(* CODESYS project std12k5_8.project

Project tree, tasks and I/O mapping:
  K1 : ELNA PLC-03-02R, OOO ELNA, version 3.5.0.31
    application std12k5
      libraries: Standard, * (System); Util, * (System); CmpSchedule, 3.5.2.0 (System); CmpLog, 3.5.2.0 (System); SysCom, 3.3.2.50 (System); SysFile, 3.3.2.50 (System); SysFileAsync, 3.3.2.50 (System); SysDir, 3.3.2.50 (System); SysTimeRtc, 3.5.0.0 (System); SysTime, 3.4.1.20 (System); CAA Storage, 3.4.4.0 (CAA Technical Workgroup); SysTypes, 3.1.2.0 (System); CmpErrors Interfaces, * (System); CmpDynamicText, 3.4.1.0 (System); SysShm, 3.3.2.50 (System); SysProcess, 3.3.2.50 (System); CmpTraceMgr, 3.5.0.0 (System); 3S Storage, 3.4.4.0 (3S - Smart Software Solutions GmbH)
      task Task (cyclic, interval t#200ms, priority 1) calls MAIN
      task TaskREZ (cyclic, interval t#110ms, priority 10) calls REZERV1
      hardwareConfig/
        data type AOConfig
        defines/
          global variables hwC
        data type DOConfig
        data type AiConfig
        data type DiConfig
      logicConfig/
        defines/
          global variables logicConfig
      program MAIN [ST]
      algoritms/
        defines/
          global variables algoritmsConf
        data type AlgoritmsConfig
        data type ImConfig
        data type ModeGpa
        data type ProtectionsConfig
        data type YstavkiConfig
      modbus/
        data type MbsConfig
        function block tstModbus [ST]: ProcessInputs, ProcessOutputs
      function block AlgoritmsManager [ST]: onStart, onInit, setMode, resetAndDisable
      function block ProtectionManager [ST]: anyProtectionSignaling
      Elpk_03_02/
        program MainUP_PRG [ST]
        global variables GVL_COMMON
        global variables GVL1N_REZ
        global variables GVLOPC
        declarations NVL1_REZ
      Symbols
      Logic/
        function block PPU_Init [ST]
        function block Synch_Rejims [ST]
        function block SIP_PS [ST]
        function block All_Quation_Off [ST]
        function block AI_Final [ST]: setNewSIP
        function block AI_Final_SIP [ST]: setNewSIP
      nasos/
        function block AutoAVOM [ST]: AVOMs_Vkl, reset, AVOMs_Vykl, run
        function block AutoNuAlg_2 [ST]: reset
        function block AutoNuAlg_1 [ST]: reset
        function block AutoPnsALg [ST]: reset
        function block AutoTEN [ST]: run, reset
        function block PNS_ON_MV_ON [ST]: reset
      function block OpcCommands [ST]
      ostanov/
        function block aoAlg [ST]: reset, run
        function block noAlg [ST]: reset, run
      Prov/
        function block Opressovka [ST]: reset
        function block Prov_dPmg [ST]: reset, run
        function block Prov_Pms [ST]: reset, run
        function block Test_Protections [ST]: reset, run, Run_Protection
        function Reset_ALL_P [ST]
      Pusk/
        function block puskSecond_faza_Chastotny [ST]: run, reset
        function block ppuAlg [ST]: AS_PS_Anologs, haveAlarms, reset, writeImStatus, remont, analogsNS, CK_Di, Neisp_DI
        function block puskFirst_faza1 [ST]: reset, run
        function block puskFirst_faza2 [ST]
        function block puskSecond_faza_Reactor [ST]: reset, run
        function block puskThird_faza [ST]: reset, run
      Start_ALG/
        function block Kran_6_Close [ST]: reset
        function block Kran_6_MOVE [ST]: reset, run
        function block PNS_Pusk [ST]: reset
        function block Reset_AutoAVOM [ST]: reset
        function block Reset_AutoTEN [ST]: reset
        function block Reset_Test_IM [ST]: reset
        function block Start_AutoAVOM [ST]: reset
        function block Start_AutoTEN [ST]: reset
        function block Start_ProtectionsVibr [ST]: reset
        function block Start_Prov_dPmg [ST]: reset
        function block Start_Prov_I [ST]: reset
        function block Start_Prov_k [ST]: reset
        function block Start_Prov_Pms [ST]: reset
        function block Start_Prov_V [ST]: reset
        function block Start_Pusk_AP [ST]: reset
        function block Start_Pusk_PP [ST]: reset
        function block Start_Test_IM [ST]: reset
        function block Start_NO [ST]: reset
        function block Start_AO [ST]: reset
        function block Start_Test_Pr [ST]: reset
      TestIm/
        function BlockIm [ST]
        function BlockOpcControl [ST]
        function block TestImAlg [ST]: reset, run
        function block Imit_OPC [ST]
      Narabotka/
        function block AO [ST]: readPersistent, writePersistent
        function block Avom1 [ST]: readPersistent, writePersistent
        function block Avom2 [ST]: readPersistent, writePersistent
        function block Avom3 [ST]: readPersistent, writePersistent
        function block Avom4 [ST]: readPersistent, writePersistent
        function block EO [ST]: readPersistent, writePersistent
        function block NO [ST]: readPersistent, writePersistent
        function block nu1 [ST]: readPersistent, writePersistent
        function block nu2 [ST]: readPersistent, writePersistent
        function block pns_ [ST]: readPersistent, writePersistent
        function block Pusk [ST]: readPersistent, writePersistent
        function block Work [ST]: readPersistent, writePersistent
        function block CMN_ [ST]: readPersistent, writePersistent
        function block Kalorifer_AVOM_ [ST]: readPersistent, writePersistent
        function block TEN_Kollectora_ [ST]: readPersistent, writePersistent
        function block TEN_MB_ [ST]: readPersistent, writePersistent
      Ystavki/
        function block AutoPNS_YT [ST]: readPersistent, writePersistent
        function block Number_Of_AVOM [ST]: writePersistent, readPersistent
        function block AutoTEN_YP [ST]: readPersistent, writePersistent
        function block AutoTEN_YT [ST]: readPersistent, writePersistent
        function block Delta_Vykl_AVOM1 [ST]: readPersistent, writePersistent
        function block Delta_Vykl_AVOM2 [ST]: readPersistent, writePersistent
        function block Delta_Vykl_AVOM3 [ST]: readPersistent, writePersistent
        function block Delta_Vykl_AVOM4 [ST]: readPersistent, writePersistent
        function block T1_AVOM [ST]: readPersistent, writePersistent
        function block T2_AVOM [ST]: readPersistent, writePersistent
        function block T3_AVOM [ST]: readPersistent, writePersistent
        function block T4_AVOM [ST]: readPersistent, writePersistent
        function block Tvkl_AVOM1 [ST]: readPersistent, writePersistent
        function block Tvkl_AVOM2 [ST]: readPersistent, writePersistent
        function block Tvkl_AVOM3 [ST]: readPersistent, writePersistent
        function block Tvkl_AVOM4 [ST]: readPersistent, writePersistent
        function block Tvykl_AVOM1 [ST]: readPersistent, writePersistent
        function block Tvykl_AVOM2 [ST]: readPersistent, writePersistent
        function block Tvykl_AVOM3 [ST]: readPersistent, writePersistent
        function block Tvykl_AVOM4 [ST]: readPersistent, writePersistent
        function block SIp_Yst [ST]: readPersistent, writePersistent
        function block AutoPNS_YP [ST]: readPersistent, writePersistent
    ADC16_15 : ADC16, OOO ELNA, version 3.5.0.31
        input  std12k5.AI_K[0].In : WORD  // In.IoData.IoData[0]
        input  std12k5.AI_K[1].In : WORD  // In.IoData.IoData[1]
        input  std12k5.AI_K[2].In : WORD  // In.IoData.IoData[2]
        input  std12k5.AI_K[3].In : WORD  // In.IoData.IoData[3]
        input  std12k5.AI_K[4].In : WORD  // In.IoData.IoData[4]
        input  std12k5.AI_K[5].In : WORD  // In.IoData.IoData[5]
        input  std12k5.AI_K[6].In : WORD  // In.IoData.IoData[6]
        input  std12k5.AI_K[7].In : WORD  // In.IoData.IoData[7]
        input  std12k5.AI_K[8].In : WORD  // In.IoData.IoData[8]
        input  std12k5.AI_K[9].In : WORD  // In.IoData.IoData[9]
        input  std12k5.AI_K[10].In : WORD  // In.IoData.IoData[10]
        input  std12k5.AI_K[11].In : WORD  // In.IoData.IoData[11]
        input  std12k5.AI_K[12].In : WORD  // In.IoData.IoData[12]
        input  std12k5.AI_K[13].In : WORD  // In.IoData.IoData[13]
        input  std12k5.AI_K[14].In : WORD  // In.IoData.IoData[14]
        input  std12k5.AI_K[15].In : WORD  // In.IoData.IoData[15]
        input  std12k5.AI_K[0].Vera : WORD  // Diagnosis.Flags.Veracity
        input  std12k5.MODULES03[15].CH_MODCONF : WORD  // Diagnosis.Service.Service[0]
        input  std12k5.MODULES03[15].CH_ERRNOW : WORD  // Diagnosis.Service.Service[1]
        input  std12k5.MODULES03[15].CH_ERRHIST : WORD  // Diagnosis.Service.Service[2]
        input  std12k5.MODULES03[15].CH_NDIAG : WORD  // Diagnosis.Service.Service[3]
        input  std12k5.MODULES03[15].CH_MDIAG : WORD  // Diagnosis.Service.Service[4]
        input  std12k5.MODULES03[15].CH_FIRMVER : WORD  // Diagnosis.Service.Service[5]
        input  std12k5.MODULES03[15].CH_FIRMDATE : WORD  // Diagnosis.Service.Service[6]
        unmapped channels: In, Diagnosis
    ADC8_14 : ADC8, OOO ELNA, version 3.5.0.31
        input  std12k5.AI_K[56].In : WORD  // In.IoData.IoData[0]
        input  std12k5.AI_K[57].In : WORD  // In.IoData.IoData[1]
        input  std12k5.AI_K[58].In : WORD  // In.IoData.IoData[2]
        input  std12k5.AI_K[59].In : WORD  // In.IoData.IoData[3]
        input  std12k5.AI_K[60].In : WORD  // In.IoData.IoData[4]
        input  std12k5.AI_K[61].In : WORD  // In.IoData.IoData[5]
        input  std12k5.AI_K[62].In : WORD  // In.IoData.IoData[6]
        input  std12k5.AI_K[63].In : WORD  // In.IoData.IoData[7]
        input  std12k5.AI_K[56].Vera : WORD  // Diagnosis.Flags.Veracity
        input  std12k5.MODULES03[14].CH_MODCONF : WORD  // Diagnosis.Service.Service[0]
        input  std12k5.MODULES03[14].CH_ERRNOW : WORD  // Diagnosis.Service.Service[1]
        input  std12k5.MODULES03[14].CH_ERRHIST : WORD  // Diagnosis.Service.Service[2]
        input  std12k5.MODULES03[14].CH_NDIAG : WORD  // Diagnosis.Service.Service[3]
        input  std12k5.MODULES03[14].CH_MDIAG : WORD  // Diagnosis.Service.Service[4]
        input  std12k5.MODULES03[14].CH_FIRMVER : WORD  // Diagnosis.Service.Service[5]
        input  std12k5.MODULES03[14].CH_FIRMDATE : WORD  // Diagnosis.Service.Service[6]
        unmapped channels: In, Diagnosis
    ADC16_13 : ADC16, OOO ELNA, version 3.5.0.31
        input  std12k5.AI_K[16].In : WORD  // In.IoData.IoData[0]
        input  std12k5.AI_K[17].In : WORD  // In.IoData.IoData[1]
        input  std12k5.AI_K[18].In : WORD  // In.IoData.IoData[2]
        input  std12k5.AI_K[19].In : WORD  // In.IoData.IoData[3]
        input  std12k5.AI_K[20].In : WORD  // In.IoData.IoData[4]
        input  std12k5.AI_K[21].In : WORD  // In.IoData.IoData[5]
        input  std12k5.AI_K[22].In : WORD  // In.IoData.IoData[6]
        input  std12k5.AI_K[23].In : WORD  // In.IoData.IoData[7]
        input  std12k5.AI_K[24].In : WORD  // In.IoData.IoData[8]
        input  std12k5.AI_K[25].In : WORD  // In.IoData.IoData[9]
        input  std12k5.AI_K[26].In : WORD  // In.IoData.IoData[10]
        input  std12k5.AI_K[27].In : WORD  // In.IoData.IoData[11]
        input  std12k5.AI_K[28].In : WORD  // In.IoData.IoData[12]
        input  std12k5.AI_K[29].In : WORD  // In.IoData.IoData[13]
        input  std12k5.AI_K[30].In : WORD  // In.IoData.IoData[14]
        input  std12k5.AI_K[31].In : WORD  // In.IoData.IoData[15]
        input  std12k5.AI_K[16].Vera : WORD  // Diagnosis.Flags.Veracity
        input  std12k5.MODULES03[13].CH_MODCONF : WORD  // Diagnosis.Service.Service[0]
        input  std12k5.MODULES03[13].CH_ERRNOW : WORD  // Diagnosis.Service.Service[1]
        input  std12k5.MODULES03[13].CH_ERRHIST : WORD  // Diagnosis.Service.Service[2]
        input  std12k5.MODULES03[13].CH_NDIAG : WORD  // Diagnosis.Service.Service[3]
        input  std12k5.MODULES03[13].CH_MDIAG : WORD  // Diagnosis.Service.Service[4]
        input  std12k5.MODULES03[13].CH_FIRMVER : WORD  // Diagnosis.Service.Service[5]
        input  std12k5.MODULES03[13].CH_FIRMDATE : WORD  // Diagnosis.Service.Service[6]
        unmapped channels: In, Diagnosis
    ADC8_12 : ADC8, OOO ELNA, version 3.5.0.31
        input  std12k5.AI_K[64].In : WORD  // In.IoData.IoData[0]
        input  std12k5.AI_K[65].In : WORD  // In.IoData.IoData[1]
        input  std12k5.AI_K[66].In : WORD  // In.IoData.IoData[2]
        input  std12k5.AI_K[67].In : WORD  // In.IoData.IoData[3]
        input  std12k5.AI_K[68].In : WORD  // In.IoData.IoData[4]
        input  std12k5.AI_K[69].In : WORD  // In.IoData.IoData[5]
        input  std12k5.AI_K[70].In : WORD  // In.IoData.IoData[6]
        input  std12k5.AI_K[71].In : WORD  // In.IoData.IoData[7]
        input  std12k5.AI_K[64].Vera : WORD  // Diagnosis.Flags.Veracity
        input  std12k5.MODULES03[12].CH_MODCONF : WORD  // Diagnosis.Service.Service[0]
        input  std12k5.MODULES03[12].CH_ERRNOW : WORD  // Diagnosis.Service.Service[1]
        input  std12k5.MODULES03[12].CH_ERRHIST : WORD  // Diagnosis.Service.Service[2]
        input  std12k5.MODULES03[12].CH_NDIAG : WORD  // Diagnosis.Service.Service[3]
        input  std12k5.MODULES03[12].CH_MDIAG : WORD  // Diagnosis.Service.Service[4]
        input  std12k5.MODULES03[12].CH_FIRMVER : WORD  // Diagnosis.Service.Service[5]
        input  std12k5.MODULES03[12].CH_FIRMDATE : WORD  // Diagnosis.Service.Service[6]
        unmapped channels: In, Diagnosis
    ADC8_11 : ADC8, OOO ELNA, version 3.5.0.31
        input  std12k5.AI_K[32].In : WORD  // In.IoData.IoData[0]
        input  std12k5.AI_K[33].In : WORD  // In.IoData.IoData[1]
        input  std12k5.AI_K[34].In : WORD  // In.IoData.IoData[2]
        input  std12k5.AI_K[35].In : WORD  // In.IoData.IoData[3]
        input  std12k5.AI_K[36].In : WORD  // In.IoData.IoData[4]
        input  std12k5.AI_K[37].In : WORD  // In.IoData.IoData[5]
        input  std12k5.AI_K[38].In : WORD  // In.IoData.IoData[6]
        input  std12k5.AI_K[39].In : WORD  // In.IoData.IoData[7]
        input  std12k5.AI_K[32].Vera : WORD  // Diagnosis.Flags.Veracity
        input  std12k5.MODULES03[11].CH_MODCONF : WORD  // Diagnosis.Service.Service[0]
        input  std12k5.MODULES03[11].CH_ERRNOW : WORD  // Diagnosis.Service.Service[1]
        input  std12k5.MODULES03[11].CH_ERRHIST : WORD  // Diagnosis.Service.Service[2]
        input  std12k5.MODULES03[11].CH_NDIAG : WORD  // Diagnosis.Service.Service[3]
        input  std12k5.MODULES03[11].CH_MDIAG : WORD  // Diagnosis.Service.Service[4]
        input  std12k5.MODULES03[11].CH_FIRMVER : WORD  // Diagnosis.Service.Service[5]
        input  std12k5.MODULES03[11].CH_FIRMDATE : WORD  // Diagnosis.Service.Service[6]
        unmapped channels: In, Diagnosis
    DIN16_10 : DIN16, OOO ELNA, version 3.5.0.31
        input  std12k5.DI_K[15].In : WORD  // In.IoData
        input  std12k5.DI_K[15].Vera : WORD  // Diagnosis.Flags.Veracity
        input  std12k5.MODULES03[10].CH_MODCONF : WORD  // Diagnosis.Service.Service[0]
        input  std12k5.MODULES03[10].CH_ERRNOW : WORD  // Diagnosis.Service.Service[1]
        input  std12k5.MODULES03[10].CH_ERRHIST : WORD  // Diagnosis.Service.Service[2]
        input  std12k5.MODULES03[10].CH_NDIAG : WORD  // Diagnosis.Service.Service[3]
        input  std12k5.MODULES03[10].CH_MDIAG : WORD  // Diagnosis.Service.Service[4]
        input  std12k5.MODULES03[10].CH_FIRMVER : WORD  // Diagnosis.Service.Service[5]
        input  std12k5.MODULES03[10].CH_FIRMDATE : WORD  // Diagnosis.Service.Service[6]
        unmapped channels: In, Diagnosis
    ADC8_9 : ADC8, OOO ELNA, version 3.5.0.31
        input  std12k5.AI_K[40].In : WORD  // In.IoData.IoData[0]
        input  std12k5.AI_K[41].In : WORD  // In.IoData.IoData[1]
        input  std12k5.AI_K[42].In : WORD  // In.IoData.IoData[2]
        input  std12k5.AI_K[43].In : WORD  // In.IoData.IoData[3]
        input  std12k5.AI_K[44].In : WORD  // In.IoData.IoData[4]
        input  std12k5.AI_K[45].In : WORD  // In.IoData.IoData[5]
        input  std12k5.AI_K[46].In : WORD  // In.IoData.IoData[6]
        input  std12k5.AI_K[47].In : WORD  // In.IoData.IoData[7]
        input  std12k5.AI_K[40].Vera : WORD  // Diagnosis.Flags.Veracity
        input  std12k5.MODULES03[9].CH_MODCONF : WORD  // Diagnosis.Service.Service[0]
        input  std12k5.MODULES03[9].CH_ERRNOW : WORD  // Diagnosis.Service.Service[1]
        input  std12k5.MODULES03[9].CH_ERRHIST : WORD  // Diagnosis.Service.Service[2]
        input  std12k5.MODULES03[9].CH_NDIAG : WORD  // Diagnosis.Service.Service[3]
        input  std12k5.MODULES03[9].CH_MDIAG : WORD  // Diagnosis.Service.Service[4]
        input  std12k5.MODULES03[9].CH_FIRMVER : WORD  // Diagnosis.Service.Service[5]
        input  std12k5.MODULES03[9].CH_FIRMDATE : WORD  // Diagnosis.Service.Service[6]
        unmapped channels: In, Diagnosis
    ADC8_16 : ADC8, OOO ELNA, version 3.5.0.31
        input  std12k5.AI_K[48].In : WORD  // In.IoData.IoData[0]
        input  std12k5.AI_K[49].In : WORD  // In.IoData.IoData[1]
        input  std12k5.AI_K[50].In : WORD  // In.IoData.IoData[2]
        input  std12k5.AI_K[51].In : WORD  // In.IoData.IoData[3]
        input  std12k5.AI_K[52].In : WORD  // In.IoData.IoData[4]
        input  std12k5.AI_K[53].In : WORD  // In.IoData.IoData[5]
        input  std12k5.AI_K[54].In : WORD  // In.IoData.IoData[6]
        input  std12k5.AI_K[55].In : WORD  // In.IoData.IoData[7]
        input  std12k5.AI_K[48].Vera : WORD  // Diagnosis.Flags.Veracity
        input  std12k5.MODULES03[16].CH_MODCONF : WORD  // Diagnosis.Service.Service[0]
        input  std12k5.MODULES03[16].CH_ERRNOW : WORD  // Diagnosis.Service.Service[1]
        input  std12k5.MODULES03[16].CH_ERRHIST : WORD  // Diagnosis.Service.Service[2]
        input  std12k5.MODULES03[16].CH_NDIAG : WORD  // Diagnosis.Service.Service[3]
        input  std12k5.MODULES03[16].CH_MDIAG : WORD  // Diagnosis.Service.Service[4]
        input  std12k5.MODULES03[16].CH_FIRMVER : WORD  // Diagnosis.Service.Service[5]
        input  std12k5.MODULES03[16].CH_FIRMDATE : WORD  // Diagnosis.Service.Service[6]
        unmapped channels: In, Diagnosis
    DIN16_8AV : DIN16, OOO ELNA, version 3.5.0.31
        input  std12k5.DI_K[14].In : WORD  // In.IoData
        input  std12k5.DI_K[14].Vera : WORD  // Diagnosis.Flags.Veracity
        input  std12k5.MODULES03[8].CH_MODCONF : WORD  // Diagnosis.Service.Service[0]
        input  std12k5.MODULES03[8].CH_ERRNOW : WORD  // Diagnosis.Service.Service[1]
        input  std12k5.MODULES03[8].CH_ERRHIST : WORD  // Diagnosis.Service.Service[2]
        input  std12k5.MODULES03[8].CH_NDIAG : WORD  // Diagnosis.Service.Service[3]
        input  std12k5.MODULES03[8].CH_MDIAG : WORD  // Diagnosis.Service.Service[4]
        input  std12k5.MODULES03[8].CH_FIRMVER : WORD  // Diagnosis.Service.Service[5]
        input  std12k5.MODULES03[8].CH_FIRMDATE : WORD  // Diagnosis.Service.Service[6]
        unmapped channels: In, Diagnosis
    DOUT16_7 : DOUT16, OOO ELNA, version 3.5.0.31
        output std12k5.DO_K[1].Q : WORD  // Out.IoData
        input  std12k5.DO_K[1].Vera : WORD  // Diagnosis.Flags.Veracity
        input  std12k5.MODULES03[7].CH_MODCONF : WORD  // Diagnosis.Service.Service[0]
        input  std12k5.MODULES03[7].CH_ERRNOW : WORD  // Diagnosis.Service.Service[1]
        input  std12k5.MODULES03[7].CH_ERRHIST : WORD  // Diagnosis.Service.Service[2]
        input  std12k5.MODULES03[7].CH_NDIAG : WORD  // Diagnosis.Service.Service[3]
        input  std12k5.MODULES03[7].CH_MDIAG : WORD  // Diagnosis.Service.Service[4]
        input  std12k5.MODULES03[7].CH_FIRMVER : WORD  // Diagnosis.Service.Service[5]
        input  std12k5.MODULES03[7].CH_FIRMDATE : WORD  // Diagnosis.Service.Service[6]
        unmapped channels: Out, Diagnosis
    DOUT16_6 : DOUT16, OOO ELNA, version 3.5.0.31
        output std12k5.DO_K[4].Q : WORD  // Out.IoData
        input  std12k5.DO_K[4].Vera : WORD  // Diagnosis.Flags.Veracity
        input  std12k5.MODULES03[6].CH_MODCONF : WORD  // Diagnosis.Service.Service[0]
        input  std12k5.MODULES03[6].CH_ERRNOW : WORD  // Diagnosis.Service.Service[1]
        input  std12k5.MODULES03[6].CH_ERRHIST : WORD  // Diagnosis.Service.Service[2]
        input  std12k5.MODULES03[6].CH_NDIAG : WORD  // Diagnosis.Service.Service[3]
        input  std12k5.MODULES03[6].CH_MDIAG : WORD  // Diagnosis.Service.Service[4]
        input  std12k5.MODULES03[6].CH_FIRMVER : WORD  // Diagnosis.Service.Service[5]
        input  std12k5.MODULES03[6].CH_FIRMDATE : WORD  // Diagnosis.Service.Service[6]
        unmapped channels: Out, Diagnosis
    DOUT16_5 : DOUT16, OOO ELNA, version 3.5.0.31
        output std12k5.DO_K[0].Q : WORD  // Out.IoData
        input  std12k5.DO_K[0].Vera : WORD  // Diagnosis.Flags.Veracity
        input  std12k5.MODULES03[5].CH_MODCONF : WORD  // Diagnosis.Service.Service[0]
        input  std12k5.MODULES03[5].CH_ERRNOW : WORD  // Diagnosis.Service.Service[1]
        input  std12k5.MODULES03[5].CH_ERRHIST : WORD  // Diagnosis.Service.Service[2]
        input  std12k5.MODULES03[5].CH_NDIAG : WORD  // Diagnosis.Service.Service[3]
        input  std12k5.MODULES03[5].CH_MDIAG : WORD  // Diagnosis.Service.Service[4]
        input  std12k5.MODULES03[5].CH_FIRMVER : WORD  // Diagnosis.Service.Service[5]
        input  std12k5.MODULES03[5].CH_FIRMDATE : WORD  // Diagnosis.Service.Service[6]
        unmapped channels: Out, Diagnosis
    DOUT16_4 : DOUT16, OOO ELNA, version 3.5.0.31
        output std12k5.DO_K[3].Q : WORD  // Out.IoData
        input  std12k5.DO_K[3].Vera : WORD  // Diagnosis.Flags.Veracity
        input  std12k5.MODULES03[4].CH_MODCONF : WORD  // Diagnosis.Service.Service[0]
        input  std12k5.MODULES03[4].CH_ERRNOW : WORD  // Diagnosis.Service.Service[1]
        input  std12k5.MODULES03[4].CH_ERRHIST : WORD  // Diagnosis.Service.Service[2]
        input  std12k5.MODULES03[4].CH_NDIAG : WORD  // Diagnosis.Service.Service[3]
        input  std12k5.MODULES03[4].CH_MDIAG : WORD  // Diagnosis.Service.Service[4]
        input  std12k5.MODULES03[4].CH_FIRMVER : WORD  // Diagnosis.Service.Service[5]
        input  std12k5.MODULES03[4].CH_FIRMDATE : WORD  // Diagnosis.Service.Service[6]
        unmapped channels: Out, Diagnosis
    MXDOUT_3 : MXDOUT, OOO ELNA, version 3.5.0.31
        input  std12k5.MODULES03[3].CH_MODCONF : WORD  // Diagnosis.Service.Service[0]
        input  std12k5.MODULES03[3].CH_ERRNOW : WORD  // Diagnosis.Service.Service[1]
        input  std12k5.MODULES03[3].CH_ERRHIST : WORD  // Diagnosis.Service.Service[2]
        input  std12k5.MODULES03[3].CH_NDIAG : WORD  // Diagnosis.Service.Service[3]
        input  std12k5.MODULES03[3].CH_MDIAG : WORD  // Diagnosis.Service.Service[4]
        input  std12k5.MODULES03[3].CH_FIRMVER : WORD  // Diagnosis.Service.Service[5]
        input  std12k5.MODULES03[3].CH_FIRMDATE : WORD  // Diagnosis.Service.Service[6]
        unmapped channels: Diagnosis
    DOUT16_2 : DOUT16, OOO ELNA, version 3.5.0.31
        output std12k5.DO_K[2].Q : WORD  // Out.IoData
        input  std12k5.DO_K[2].Vera : WORD  // Diagnosis.Flags.Veracity
        input  std12k5.MODULES03[2].CH_MODCONF : WORD  // Diagnosis.Service.Service[0]
        input  std12k5.MODULES03[2].CH_ERRNOW : WORD  // Diagnosis.Service.Service[1]
        input  std12k5.MODULES03[2].CH_ERRHIST : WORD  // Diagnosis.Service.Service[2]
        input  std12k5.MODULES03[2].CH_NDIAG : WORD  // Diagnosis.Service.Service[3]
        input  std12k5.MODULES03[2].CH_MDIAG : WORD  // Diagnosis.Service.Service[4]
        input  std12k5.MODULES03[2].CH_FIRMVER : WORD  // Diagnosis.Service.Service[5]
        input  std12k5.MODULES03[2].CH_FIRMDATE : WORD  // Diagnosis.Service.Service[6]
        unmapped channels: Out, Diagnosis
    MXDIN_1 : MXDIN, OOO ELNA, version 3.5.0.31
        input  std12k5.DI_K[0].In : WORD  // In.IoData.IoData[0]
        input  std12k5.DI_K[1].In : WORD  // In.IoData.IoData[1]
        input  std12k5.DI_K[2].In : WORD  // In.IoData.IoData[2]
        input  std12k5.DI_K[3].In : WORD  // In.IoData.IoData[3]
        input  std12k5.DI_K[4].In : WORD  // In.IoData.IoData[4]
        input  std12k5.DI_K[5].In : WORD  // In.IoData.IoData[5]
        input  std12k5.DI_K[6].In : WORD  // In.IoData.IoData[6]
        input  std12k5.DI_K[7].In : WORD  // In.IoData.IoData[7]
        input  std12k5.DI_K[8].In : WORD  // In.IoData.IoData[8]
        input  std12k5.DI_K[9].In : WORD  // In.IoData.IoData[9]
        input  std12k5.DI_K[10].In : WORD  // In.IoData.IoData[10]
        input  std12k5.DI_K[11].In : WORD  // In.IoData.IoData[11]
        input  std12k5.DI_K[12].In : WORD  // In.IoData.IoData[12]
        input  std12k5.DI_K[13].In : WORD  // In.IoData.IoData[13]
        input  std12k5.DI_K[0].Vera : WORD  // Diagnosis.Flags.Veracity
        input  std12k5.MODULES03[1].CH_MODCONF : WORD  // Diagnosis.Service.Service[0]
        input  std12k5.MODULES03[1].CH_ERRNOW : WORD  // Diagnosis.Service.Service[1]
        input  std12k5.MODULES03[1].CH_ERRHIST : WORD  // Diagnosis.Service.Service[2]
        input  std12k5.MODULES03[1].CH_NDIAG : WORD  // Diagnosis.Service.Service[3]
        input  std12k5.MODULES03[1].CH_MDIAG : WORD  // Diagnosis.Service.Service[4]
        input  std12k5.MODULES03[1].CH_FIRMVER : WORD  // Diagnosis.Service.Service[5]
        input  std12k5.MODULES03[1].CH_FIRMDATE : WORD  // Diagnosis.Service.Service[6]
        unmapped channels: In, Diagnosis
    Virtual_IO : Virtual IO, OOO ELNA, version 3.5.0.31
        output std12k5.MxMode_O : WORD  // Main Service Outputs.MXMODE
        output std12k5.MainUP_PRG.ADCWAY_O : WORD  // Main Service Outputs.ADCWAY
        output std12k5.MainUP_PRG.HIDE_ERR_OUT_O : WORD  // Main Service Outputs.HIDE_ERR_OUT
        output std12k5.MainUP_PRG.WDOG_O : WORD  // Main Service Outputs.WDOG
        input  std12k5.MxStatus_I : WORD  // Main Service Inputs.MXSTAT
        input  std12k5.MainUP_PRG.ADCWAY_I : WORD  // Main Service Inputs.ADCWAY
        input  std12k5.BMPPRES_I : WORD  // Main Service Inputs.BMPPRES
        input  std12k5.BMPERR_I : WORD  // Main Service Inputs.BMPERR
        input  std12k5.MainUP_PRG.MXLINES_I : WORD  // Main Service Inputs.MXLINES
        input  std12k5.MainUP_PRG.HIDE_ERR_OUT_I : WORD  // Main Service Inputs.HIDE_ERR_OUT
        input  std12k5.MainUP_PRG.RWH_PERIOD_I : WORD  // Main Service Inputs.RWH_PERIOD
        input  std12k5.MainUP_PRG.MX_ATT_I : WORD  // Main Service Inputs.MX_ATT
        input  std12k5.MainUP_PRG.EXTCMD_I : WORD  // Main Service Inputs.EXTCMD
        unmapped channels: Main Service Outputs, Main Service Inputs, ComPort Outputs, ComPort Inputs, Redundancy Inputs
  K2 : ELNA PLC-03-02R, OOO ELNA, version 3.5.0.31
    application std12k5
      libraries: Standard, * (System); Util, * (System); CmpSchedule, 3.5.2.0 (System); CmpLog, 3.5.2.0 (System); SysCom, 3.3.2.50 (System); SysFile, 3.3.2.50 (System); SysFileAsync, 3.3.2.50 (System); SysDir, 3.3.2.50 (System); SysTimeRtc, 3.5.0.0 (System); SysTime, 3.4.1.20 (System); CAA Storage, 3.4.4.0 (CAA Technical Workgroup); SysTypes, 3.1.2.0 (System); CmpErrors Interfaces, * (System); CmpDynamicText, 3.4.1.0 (System); SysShm, 3.3.2.50 (System); SysProcess, 3.3.2.50 (System); CmpTraceMgr, 3.5.0.0 (System); 3S Storage, 3.4.4.0 (3S - Smart Software Solutions GmbH)
      task Task (cyclic, interval t#200ms, priority 1) calls MAIN
      task TaskREZ (cyclic, interval t#110ms, priority 10) calls REZERV2
      hardwareConfig/
        defines/
          global variables hwC
        data type AOConfig
        data type DOConfig
        data type AiConfig
        data type DiConfig
      logicConfig/
        defines/
          global variables logicConfig
      program MAIN [ST]
      algoritms/
        defines/
          global variables algoritmsConf
        data type AlgoritmsConfig
        data type ModeGpa
        data type ProtectionsConfig
        data type ImConfig
        data type YstavkiConfig
      function block AlgoritmsManager [ST]: onStart, onInit, setMode, resetAndDisable
      function block ProtectionManager [ST]: anyProtectionSignaling
      modbus/
        data type MbsConfig
        function block tstModbus [ST]: ProcessInputs, ProcessOutputs
      Elpk_03_02/
        program MainUP_PRG [ST]
        global variables GVL_COMMON
        global variables GVL2N_REZ
        global variables GVLOPC
        declarations NVL2_REZ
      Symbols
      Logic/
        function block AI_Final [ST]: setNewSIP
        function block SIP_PS [ST]
        function block Synch_Rejims [ST]
        function block All_Quation_Off [ST]
        function block PPU_Init [ST]
        function block AI_Final_SIP [ST]: setNewSIP
      Pusk/
        function block puskSecond_faza_Chastotny [ST]: reset, run
        function block ppuAlg [ST]: Neisp_DI, analogsNS, AS_PS_Anologs, haveAlarms, reset, writeImStatus, CK_Di, remont
        function block puskFirst_faza1 [ST]: reset, run
        function block puskFirst_faza2 [ST]
        function block puskSecond_faza_Reactor [ST]: reset, run
        function block puskThird_faza [ST]: reset, run
      nasos/
        function block AutoAVOM [ST]: AVOMs_Vkl, reset, AVOMs_Vykl, run
        function block AutoNuAlg_2 [ST]: reset
        function block AutoNuAlg_1 [ST]: reset
        function block AutoPnsALg [ST]: reset
        function block AutoTEN [ST]: run, reset
        function block PNS_ON_MV_ON [ST]: reset
      function block OpcCommands [ST]
      ostanov/
        function block aoAlg [ST]: reset, run
        function block noAlg [ST]: reset, run
      Prov/
        function block Opressovka [ST]: reset
        function block Prov_dPmg [ST]: reset, run
        function block Prov_Pms [ST]: reset, run
        function Reset_ALL_P [ST]
        function block Test_Protections [ST]: reset, run, Run_Protection
      Start_ALG/
        function block Kran_6_Close [ST]: reset
        function block Kran_6_MOVE [ST]: reset, run
        function block PNS_Pusk [ST]: reset
        function block Reset_AutoAVOM [ST]: reset
        function block Reset_AutoTEN [ST]: reset
        function block Reset_Test_IM [ST]: reset
        function block Start_AutoAVOM [ST]: reset
        function block Start_AutoTEN [ST]: reset
        function block Start_ProtectionsVibr [ST]: reset
        function block Start_Prov_dPmg [ST]: reset
        function block Start_Prov_I [ST]: reset
        function block Start_Prov_k [ST]: reset
        function block Start_Prov_Pms [ST]: reset
        function block Start_Prov_V [ST]: reset
        function block Start_Pusk_AP [ST]: reset
        function block Start_Pusk_PP [ST]: reset
        function block Start_Test_IM [ST]: reset
        function block Start_NO [ST]: reset
        function block Start_AO [ST]: reset
        function block Start_Test_Pr [ST]: reset
      TestIm/
        function BlockIm [ST]
        function BlockOpcControl [ST]
        function block TestImAlg [ST]: reset, run
        function block Imit_OPC [ST]
      Natabotka/
        function block AO [ST]: readPersistent, writePersistent
        function block Avom1 [ST]: readPersistent, writePersistent
        function block Avom2 [ST]: readPersistent, writePersistent
        function block Avom3 [ST]: readPersistent, writePersistent
        function block Avom4 [ST]: readPersistent, writePersistent
        function block EO [ST]: readPersistent, writePersistent
        function block NO [ST]: readPersistent, writePersistent
        function block nu1 [ST]: readPersistent, writePersistent
        function block nu2 [ST]: readPersistent, writePersistent
        function block pns_ [ST]: readPersistent, writePersistent
        function block Pusk [ST]: readPersistent, writePersistent
        function block Work [ST]: readPersistent, writePersistent
        function block CMN_ [ST]: readPersistent, writePersistent
        function block Kalorifer_AVOM_ [ST]: readPersistent, writePersistent
        function block TEN_Kollectora_ [ST]: readPersistent, writePersistent
        function block TEN_MB_ [ST]: readPersistent, writePersistent
      Ystavki/
        function block AutoPNS_YP [ST]: readPersistent, writePersistent
        function block Number_Of_AVOM [ST]: writePersistent, readPersistent
        function block AutoPNS_YT [ST]: readPersistent, writePersistent
        function block AutoTEN_YP [ST]: readPersistent, writePersistent
        function block AutoTEN_YT [ST]: readPersistent, writePersistent
        function block Delta_Vykl_AVOM1 [ST]: readPersistent, writePersistent
        function block Delta_Vykl_AVOM2 [ST]: readPersistent, writePersistent
        function block Delta_Vykl_AVOM3 [ST]: readPersistent, writePersistent
        function block Delta_Vykl_AVOM4 [ST]: readPersistent, writePersistent
        function block T1_AVOM [ST]: readPersistent, writePersistent
        function block T2_AVOM [ST]: readPersistent, writePersistent
        function block T3_AVOM [ST]: readPersistent, writePersistent
        function block T4_AVOM [ST]: readPersistent, writePersistent
        function block Tvkl_AVOM1 [ST]: readPersistent, writePersistent
        function block Tvkl_AVOM2 [ST]: readPersistent, writePersistent
        function block Tvkl_AVOM3 [ST]: readPersistent, writePersistent
        function block Tvkl_AVOM4 [ST]: readPersistent, writePersistent
        function block Tvykl_AVOM1 [ST]: readPersistent, writePersistent
        function block Tvykl_AVOM2 [ST]: readPersistent, writePersistent
        function block Tvykl_AVOM3 [ST]: readPersistent, writePersistent
        function block Tvykl_AVOM4 [ST]: readPersistent, writePersistent
        function block SIp_Yst [ST]: readPersistent, writePersistent
    Virtual_IO : Virtual IO, OOO ELNA, version 3.5.0.31
        output std12k5.MxMode_O : WORD  // Main Service Outputs.MXMODE
        output std12k5.MainUP_PRG.ADCWAY_O : WORD  // Main Service Outputs.ADCWAY
        output std12k5.MainUP_PRG.HIDE_ERR_OUT_O : WORD  // Main Service Outputs.HIDE_ERR_OUT
        output std12k5.MainUP_PRG.WDOG_O : WORD  // Main Service Outputs.WDOG
        input  std12k5.MxStatus_I : WORD  // Main Service Inputs.MXSTAT
        input  std12k5.MainUP_PRG.ADCWAY_I : WORD  // Main Service Inputs.ADCWAY
        input  std12k5.BMPPRES_I : WORD  // Main Service Inputs.BMPPRES
        input  std12k5.BMPERR_I : WORD  // Main Service Inputs.BMPERR
        input  std12k5.MainUP_PRG.MXLINES_I : WORD  // Main Service Inputs.MXLINES
        input  std12k5.MainUP_PRG.HIDE_ERR_OUT_I : WORD  // Main Service Inputs.HIDE_ERR_OUT
        input  std12k5.MainUP_PRG.RWH_PERIOD_I : WORD  // Main Service Inputs.RWH_PERIOD
        input  std12k5.MainUP_PRG.MX_ATT_I : WORD  // Main Service Inputs.MX_ATT
        input  std12k5.MainUP_PRG.EXTCMD_I : WORD  // Main Service Inputs.EXTCMD
        unmapped channels: Main Service Outputs, Main Service Inputs, ComPort Outputs, ComPort Inputs, Redundancy Inputs
    MXDIN_1 : MXDIN, OOO ELNA, version 3.5.0.31
        input  std12k5.DI_K[0].In : WORD  // In.IoData.IoData[0]
        input  std12k5.DI_K[1].In : WORD  // In.IoData.IoData[1]
        input  std12k5.DI_K[2].In : WORD  // In.IoData.IoData[2]
        input  std12k5.DI_K[3].In : WORD  // In.IoData.IoData[3]
        input  std12k5.DI_K[4].In : WORD  // In.IoData.IoData[4]
        input  std12k5.DI_K[5].In : WORD  // In.IoData.IoData[5]
        input  std12k5.DI_K[6].In : WORD  // In.IoData.IoData[6]
        input  std12k5.DI_K[7].In : WORD  // In.IoData.IoData[7]
        input  std12k5.DI_K[8].In : WORD  // In.IoData.IoData[8]
        input  std12k5.DI_K[9].In : WORD  // In.IoData.IoData[9]
        input  std12k5.DI_K[10].In : WORD  // In.IoData.IoData[10]
        input  std12k5.DI_K[11].In : WORD  // In.IoData.IoData[11]
        input  std12k5.DI_K[12].In : WORD  // In.IoData.IoData[12]
        input  std12k5.DI_K[13].In : WORD  // In.IoData.IoData[13]
        input  std12k5.DI_K[0].Vera : WORD  // Diagnosis.Flags.Veracity
        input  std12k5.MODULES03[1].CH_MODCONF : WORD  // Diagnosis.Service.Service[0]
        input  std12k5.MODULES03[1].CH_ERRNOW : WORD  // Diagnosis.Service.Service[1]
        input  std12k5.MODULES03[1].CH_ERRHIST : WORD  // Diagnosis.Service.Service[2]
        input  std12k5.MODULES03[1].CH_NDIAG : WORD  // Diagnosis.Service.Service[3]
        input  std12k5.MODULES03[1].CH_MDIAG : WORD  // Diagnosis.Service.Service[4]
        input  std12k5.MODULES03[1].CH_FIRMVER : WORD  // Diagnosis.Service.Service[5]
        input  std12k5.MODULES03[1].CH_FIRMDATE : WORD  // Diagnosis.Service.Service[6]
        unmapped channels: In, Diagnosis
    DOUT16_2 : DOUT16, OOO ELNA, version 3.5.0.31
        output std12k5.DO_K[2].Q : WORD  // Out.IoData
        input  std12k5.DO_K[2].Vera : WORD  // Diagnosis.Flags.Veracity
        input  std12k5.MODULES03[2].CH_MODCONF : WORD  // Diagnosis.Service.Service[0]
        input  std12k5.MODULES03[2].CH_ERRNOW : WORD  // Diagnosis.Service.Service[1]
        input  std12k5.MODULES03[2].CH_ERRHIST : WORD  // Diagnosis.Service.Service[2]
        input  std12k5.MODULES03[2].CH_NDIAG : WORD  // Diagnosis.Service.Service[3]
        input  std12k5.MODULES03[2].CH_MDIAG : WORD  // Diagnosis.Service.Service[4]
        input  std12k5.MODULES03[2].CH_FIRMVER : WORD  // Diagnosis.Service.Service[5]
        input  std12k5.MODULES03[2].CH_FIRMDATE : WORD  // Diagnosis.Service.Service[6]
        unmapped channels: Out, Diagnosis
    MXDOUT_3 : MXDOUT, OOO ELNA, version 3.5.0.31
        input  std12k5.MODULES03[3].CH_MODCONF : WORD  // Diagnosis.Service.Service[0]
        input  std12k5.MODULES03[3].CH_ERRNOW : WORD  // Diagnosis.Service.Service[1]
        input  std12k5.MODULES03[3].CH_ERRHIST : WORD  // Diagnosis.Service.Service[2]
        input  std12k5.MODULES03[3].CH_NDIAG : WORD  // Diagnosis.Service.Service[3]
        input  std12k5.MODULES03[3].CH_MDIAG : WORD  // Diagnosis.Service.Service[4]
        input  std12k5.MODULES03[3].CH_FIRMVER : WORD  // Diagnosis.Service.Service[5]
        input  std12k5.MODULES03[3].CH_FIRMDATE : WORD  // Diagnosis.Service.Service[6]
        unmapped channels: Diagnosis
    DOUT16_4 : DOUT16, OOO ELNA, version 3.5.0.31
        output std12k5.DO_K[3].Q : WORD  // Out.IoData
        input  std12k5.DO_K[3].Vera : WORD  // Diagnosis.Flags.Veracity
        input  std12k5.MODULES03[4].CH_MODCONF : WORD  // Diagnosis.Service.Service[0]
        input  std12k5.MODULES03[4].CH_ERRNOW : WORD  // Diagnosis.Service.Service[1]
        input  std12k5.MODULES03[4].CH_ERRHIST : WORD  // Diagnosis.Service.Service[2]
        input  std12k5.MODULES03[4].CH_NDIAG : WORD  // Diagnosis.Service.Service[3]
        input  std12k5.MODULES03[4].CH_MDIAG : WORD  // Diagnosis.Service.Service[4]
        input  std12k5.MODULES03[4].CH_FIRMVER : WORD  // Diagnosis.Service.Service[5]
        input  std12k5.MODULES03[4].CH_FIRMDATE : WORD  // Diagnosis.Service.Service[6]
        unmapped channels: Out, Diagnosis
    DOUT16_5 : DOUT16, OOO ELNA, version 3.5.0.31
        output std12k5.DO_K[0].Q : WORD  // Out.IoData
        input  std12k5.DO_K[0].Vera : WORD  // Diagnosis.Flags.Veracity
        input  std12k5.MODULES03[5].CH_MODCONF : WORD  // Diagnosis.Service.Service[0]
        input  std12k5.MODULES03[5].CH_ERRNOW : WORD  // Diagnosis.Service.Service[1]
        input  std12k5.MODULES03[5].CH_ERRHIST : WORD  // Diagnosis.Service.Service[2]
        input  std12k5.MODULES03[5].CH_NDIAG : WORD  // Diagnosis.Service.Service[3]
        input  std12k5.MODULES03[5].CH_MDIAG : WORD  // Diagnosis.Service.Service[4]
        input  std12k5.MODULES03[5].CH_FIRMVER : WORD  // Diagnosis.Service.Service[5]
        input  std12k5.MODULES03[5].CH_FIRMDATE : WORD  // Diagnosis.Service.Service[6]
        unmapped channels: Out, Diagnosis
    DOUT16_6 : DOUT16, OOO ELNA, version 3.5.0.31
        output std12k5.DO_K[4].Q : WORD  // Out.IoData
        input  std12k5.DO_K[4].Vera : WORD  // Diagnosis.Flags.Veracity
        input  std12k5.MODULES03[6].CH_MODCONF : WORD  // Diagnosis.Service.Service[0]
        input  std12k5.MODULES03[6].CH_ERRNOW : WORD  // Diagnosis.Service.Service[1]
        input  std12k5.MODULES03[6].CH_ERRHIST : WORD  // Diagnosis.Service.Service[2]
        input  std12k5.MODULES03[6].CH_NDIAG : WORD  // Diagnosis.Service.Service[3]
        input  std12k5.MODULES03[6].CH_MDIAG : WORD  // Diagnosis.Service.Service[4]
        input  std12k5.MODULES03[6].CH_FIRMVER : WORD  // Diagnosis.Service.Service[5]
        input  std12k5.MODULES03[6].CH_FIRMDATE : WORD  // Diagnosis.Service.Service[6]
        unmapped channels: Out, Diagnosis
    DOUT16_7 : DOUT16, OOO ELNA, version 3.5.0.31
        output std12k5.DO_K[1].Q : WORD  // Out.IoData
        input  std12k5.DO_K[1].Vera : WORD  // Diagnosis.Flags.Veracity
        input  std12k5.MODULES03[7].CH_MODCONF : WORD  // Diagnosis.Service.Service[0]
        input  std12k5.MODULES03[7].CH_ERRNOW : WORD  // Diagnosis.Service.Service[1]
        input  std12k5.MODULES03[7].CH_ERRHIST : WORD  // Diagnosis.Service.Service[2]
        input  std12k5.MODULES03[7].CH_NDIAG : WORD  // Diagnosis.Service.Service[3]
        input  std12k5.MODULES03[7].CH_MDIAG : WORD  // Diagnosis.Service.Service[4]
        input  std12k5.MODULES03[7].CH_FIRMVER : WORD  // Diagnosis.Service.Service[5]
        input  std12k5.MODULES03[7].CH_FIRMDATE : WORD  // Diagnosis.Service.Service[6]
        unmapped channels: Out, Diagnosis
    DIN16_8AV : DIN16, OOO ELNA, version 3.5.0.31
        input  std12k5.DI_K[14].In : WORD  // In.IoData
        input  std12k5.DI_K[14].Vera : WORD  // Diagnosis.Flags.Veracity
        input  std12k5.MODULES03[8].CH_MODCONF : WORD  // Diagnosis.Service.Service[0]
        input  std12k5.MODULES03[8].CH_ERRNOW : WORD  // Diagnosis.Service.Service[1]
        input  std12k5.MODULES03[8].CH_ERRHIST : WORD  // Diagnosis.Service.Service[2]
        input  std12k5.MODULES03[8].CH_NDIAG : WORD  // Diagnosis.Service.Service[3]
        input  std12k5.MODULES03[8].CH_MDIAG : WORD  // Diagnosis.Service.Service[4]
        input  std12k5.MODULES03[8].CH_FIRMVER : WORD  // Diagnosis.Service.Service[5]
        input  std12k5.MODULES03[8].CH_FIRMDATE : WORD  // Diagnosis.Service.Service[6]
        unmapped channels: In, Diagnosis
    ADC8_9 : ADC8, OOO ELNA, version 3.5.0.31
        input  std12k5.AI_K[40].In : WORD  // In.IoData.IoData[0]
        input  std12k5.AI_K[41].In : WORD  // In.IoData.IoData[1]
        input  std12k5.AI_K[42].In : WORD  // In.IoData.IoData[2]
        input  std12k5.AI_K[43].In : WORD  // In.IoData.IoData[3]
        input  std12k5.AI_K[44].In : WORD  // In.IoData.IoData[4]
        input  std12k5.AI_K[45].In : WORD  // In.IoData.IoData[5]
        input  std12k5.AI_K[46].In : WORD  // In.IoData.IoData[6]
        input  std12k5.AI_K[47].In : WORD  // In.IoData.IoData[7]
        input  std12k5.AI_K[40].Vera : WORD  // Diagnosis.Flags.Veracity
        input  std12k5.MODULES03[9].CH_MODCONF : WORD  // Diagnosis.Service.Service[0]
        input  std12k5.MODULES03[9].CH_ERRNOW : WORD  // Diagnosis.Service.Service[1]
        input  std12k5.MODULES03[9].CH_ERRHIST : WORD  // Diagnosis.Service.Service[2]
        input  std12k5.MODULES03[9].CH_NDIAG : WORD  // Diagnosis.Service.Service[3]
        input  std12k5.MODULES03[9].CH_MDIAG : WORD  // Diagnosis.Service.Service[4]
        input  std12k5.MODULES03[9].CH_FIRMVER : WORD  // Diagnosis.Service.Service[5]
        input  std12k5.MODULES03[9].CH_FIRMDATE : WORD  // Diagnosis.Service.Service[6]
        unmapped channels: In, Diagnosis
    DIN16_10 : DIN16, OOO ELNA, version 3.5.0.31
        input  std12k5.DI_K[15].In : WORD  // In.IoData
        input  std12k5.DI_K[15].Vera : WORD  // Diagnosis.Flags.Veracity
        input  std12k5.MODULES03[10].CH_MODCONF : WORD  // Diagnosis.Service.Service[0]
        input  std12k5.MODULES03[10].CH_ERRNOW : WORD  // Diagnosis.Service.Service[1]
        input  std12k5.MODULES03[10].CH_ERRHIST : WORD  // Diagnosis.Service.Service[2]
        input  std12k5.MODULES03[10].CH_NDIAG : WORD  // Diagnosis.Service.Service[3]
        input  std12k5.MODULES03[10].CH_MDIAG : WORD  // Diagnosis.Service.Service[4]
        input  std12k5.MODULES03[10].CH_FIRMVER : WORD  // Diagnosis.Service.Service[5]
        input  std12k5.MODULES03[10].CH_FIRMDATE : WORD  // Diagnosis.Service.Service[6]
        unmapped channels: In, Diagnosis
    ADC8_11 : ADC8, OOO ELNA, version 3.5.0.31
        input  std12k5.AI_K[32].In : WORD  // In.IoData.IoData[0]
        input  std12k5.AI_K[33].In : WORD  // In.IoData.IoData[1]
        input  std12k5.AI_K[34].In : WORD  // In.IoData.IoData[2]
        input  std12k5.AI_K[35].In : WORD  // In.IoData.IoData[3]
        input  std12k5.AI_K[36].In : WORD  // In.IoData.IoData[4]
        input  std12k5.AI_K[37].In : WORD  // In.IoData.IoData[5]
        input  std12k5.AI_K[38].In : WORD  // In.IoData.IoData[6]
        input  std12k5.AI_K[39].In : WORD  // In.IoData.IoData[7]
        input  std12k5.AI_K[32].Vera : WORD  // Diagnosis.Flags.Veracity
        input  std12k5.MODULES03[11].CH_MODCONF : WORD  // Diagnosis.Service.Service[0]
        input  std12k5.MODULES03[11].CH_ERRNOW : WORD  // Diagnosis.Service.Service[1]
        input  std12k5.MODULES03[11].CH_ERRHIST : WORD  // Diagnosis.Service.Service[2]
        input  std12k5.MODULES03[11].CH_NDIAG : WORD  // Diagnosis.Service.Service[3]
        input  std12k5.MODULES03[11].CH_MDIAG : WORD  // Diagnosis.Service.Service[4]
        input  std12k5.MODULES03[11].CH_FIRMVER : WORD  // Diagnosis.Service.Service[5]
        input  std12k5.MODULES03[11].CH_FIRMDATE : WORD  // Diagnosis.Service.Service[6]
        unmapped channels: In, Diagnosis
    ADC8_12 : ADC8, OOO ELNA, version 3.5.0.31
        input  std12k5.AI_K[64].In : WORD  // In.IoData.IoData[0]
        input  std12k5.AI_K[65].In : WORD  // In.IoData.IoData[1]
        input  std12k5.AI_K[66].In : WORD  // In.IoData.IoData[2]
        input  std12k5.AI_K[67].In : WORD  // In.IoData.IoData[3]
        input  std12k5.AI_K[68].In : WORD  // In.IoData.IoData[4]
        input  std12k5.AI_K[69].In : WORD  // In.IoData.IoData[5]
        input  std12k5.AI_K[70].In : WORD  // In.IoData.IoData[6]
        input  std12k5.AI_K[71].In : WORD  // In.IoData.IoData[7]
        input  std12k5.AI_K[64].Vera : WORD  // Diagnosis.Flags.Veracity
        input  std12k5.MODULES03[12].CH_MODCONF : WORD  // Diagnosis.Service.Service[0]
        input  std12k5.MODULES03[12].CH_ERRNOW : WORD  // Diagnosis.Service.Service[1]
        input  std12k5.MODULES03[12].CH_ERRHIST : WORD  // Diagnosis.Service.Service[2]
        input  std12k5.MODULES03[12].CH_NDIAG : WORD  // Diagnosis.Service.Service[3]
        input  std12k5.MODULES03[12].CH_MDIAG : WORD  // Diagnosis.Service.Service[4]
        input  std12k5.MODULES03[12].CH_FIRMVER : WORD  // Diagnosis.Service.Service[5]
        input  std12k5.MODULES03[12].CH_FIRMDATE : WORD  // Diagnosis.Service.Service[6]
        unmapped channels: In, Diagnosis
    ADC16_13 : ADC16, OOO ELNA, version 3.5.0.31
        input  std12k5.AI_K[16].In : WORD  // In.IoData.IoData[0]
        input  std12k5.AI_K[17].In : WORD  // In.IoData.IoData[1]
        input  std12k5.AI_K[18].In : WORD  // In.IoData.IoData[2]
        input  std12k5.AI_K[19].In : WORD  // In.IoData.IoData[3]
        input  std12k5.AI_K[20].In : WORD  // In.IoData.IoData[4]
        input  std12k5.AI_K[21].In : WORD  // In.IoData.IoData[5]
        input  std12k5.AI_K[22].In : WORD  // In.IoData.IoData[6]
        input  std12k5.AI_K[23].In : WORD  // In.IoData.IoData[7]
        input  std12k5.AI_K[24].In : WORD  // In.IoData.IoData[8]
        input  std12k5.AI_K[25].In : WORD  // In.IoData.IoData[9]
        input  std12k5.AI_K[26].In : WORD  // In.IoData.IoData[10]
        input  std12k5.AI_K[27].In : WORD  // In.IoData.IoData[11]
        input  std12k5.AI_K[28].In : WORD  // In.IoData.IoData[12]
        input  std12k5.AI_K[29].In : WORD  // In.IoData.IoData[13]
        input  std12k5.AI_K[30].In : WORD  // In.IoData.IoData[14]
        input  std12k5.AI_K[31].In : WORD  // In.IoData.IoData[15]
        input  std12k5.AI_K[16].Vera : WORD  // Diagnosis.Flags.Veracity
        input  std12k5.MODULES03[13].CH_MODCONF : WORD  // Diagnosis.Service.Service[0]
        input  std12k5.MODULES03[13].CH_ERRNOW : WORD  // Diagnosis.Service.Service[1]
        input  std12k5.MODULES03[13].CH_ERRHIST : WORD  // Diagnosis.Service.Service[2]
        input  std12k5.MODULES03[13].CH_NDIAG : WORD  // Diagnosis.Service.Service[3]
        input  std12k5.MODULES03[13].CH_MDIAG : WORD  // Diagnosis.Service.Service[4]
        input  std12k5.MODULES03[13].CH_FIRMVER : WORD  // Diagnosis.Service.Service[5]
        input  std12k5.MODULES03[13].CH_FIRMDATE : WORD  // Diagnosis.Service.Service[6]
        unmapped channels: In, Diagnosis
    ADC8_14 : ADC8, OOO ELNA, version 3.5.0.31
        input  std12k5.AI_K[56].In : WORD  // In.IoData.IoData[0]
        input  std12k5.AI_K[57].In : WORD  // In.IoData.IoData[1]
        input  std12k5.AI_K[58].In : WORD  // In.IoData.IoData[2]
        input  std12k5.AI_K[59].In : WORD  // In.IoData.IoData[3]
        input  std12k5.AI_K[60].In : WORD  // In.IoData.IoData[4]
        input  std12k5.AI_K[61].In : WORD  // In.IoData.IoData[5]
        input  std12k5.AI_K[62].In : WORD  // In.IoData.IoData[6]
        input  std12k5.AI_K[63].In : WORD  // In.IoData.IoData[7]
        input  std12k5.AI_K[56].Vera : WORD  // Diagnosis.Flags.Veracity
        input  std12k5.MODULES03[14].CH_MODCONF : WORD  // Diagnosis.Service.Service[0]
        input  std12k5.MODULES03[14].CH_ERRNOW : WORD  // Diagnosis.Service.Service[1]
        input  std12k5.MODULES03[14].CH_ERRHIST : WORD  // Diagnosis.Service.Service[2]
        input  std12k5.MODULES03[14].CH_NDIAG : WORD  // Diagnosis.Service.Service[3]
        input  std12k5.MODULES03[14].CH_MDIAG : WORD  // Diagnosis.Service.Service[4]
        input  std12k5.MODULES03[14].CH_FIRMVER : WORD  // Diagnosis.Service.Service[5]
        input  std12k5.MODULES03[14].CH_FIRMDATE : WORD  // Diagnosis.Service.Service[6]
        unmapped channels: In, Diagnosis
    ADC16_15 : ADC16, OOO ELNA, version 3.5.0.31
        input  std12k5.AI_K[0].In : WORD  // In.IoData.IoData[0]
        input  std12k5.AI_K[1].In : WORD  // In.IoData.IoData[1]
        input  std12k5.AI_K[2].In : WORD  // In.IoData.IoData[2]
        input  std12k5.AI_K[3].In : WORD  // In.IoData.IoData[3]
        input  std12k5.AI_K[4].In : WORD  // In.IoData.IoData[4]
        input  std12k5.AI_K[5].In : WORD  // In.IoData.IoData[5]
        input  std12k5.AI_K[6].In : WORD  // In.IoData.IoData[6]
        input  std12k5.AI_K[7].In : WORD  // In.IoData.IoData[7]
        input  std12k5.AI_K[8].In : WORD  // In.IoData.IoData[8]
        input  std12k5.AI_K[9].In : WORD  // In.IoData.IoData[9]
        input  std12k5.AI_K[10].In : WORD  // In.IoData.IoData[10]
        input  std12k5.AI_K[11].In : WORD  // In.IoData.IoData[11]
        input  std12k5.AI_K[12].In : WORD  // In.IoData.IoData[12]
        input  std12k5.AI_K[13].In : WORD  // In.IoData.IoData[13]
        input  std12k5.AI_K[14].In : WORD  // In.IoData.IoData[14]
        input  std12k5.AI_K[15].In : WORD  // In.IoData.IoData[15]
        input  std12k5.AI_K[0].Vera : WORD  // Diagnosis.Flags.Veracity
        input  std12k5.MODULES03[15].CH_MODCONF : WORD  // Diagnosis.Service.Service[0]
        input  std12k5.MODULES03[15].CH_ERRNOW : WORD  // Diagnosis.Service.Service[1]
        input  std12k5.MODULES03[15].CH_ERRHIST : WORD  // Diagnosis.Service.Service[2]
        input  std12k5.MODULES03[15].CH_NDIAG : WORD  // Diagnosis.Service.Service[3]
        input  std12k5.MODULES03[15].CH_MDIAG : WORD  // Diagnosis.Service.Service[4]
        input  std12k5.MODULES03[15].CH_FIRMVER : WORD  // Diagnosis.Service.Service[5]
        input  std12k5.MODULES03[15].CH_FIRMDATE : WORD  // Diagnosis.Service.Service[6]
        unmapped channels: In, Diagnosis
    ADC8_16 : ADC8, OOO ELNA, version 3.5.0.31
        input  std12k5.AI_K[48].In : WORD  // In.IoData.IoData[0]
        input  std12k5.AI_K[49].In : WORD  // In.IoData.IoData[1]
        input  std12k5.AI_K[50].In : WORD  // In.IoData.IoData[2]
        input  std12k5.AI_K[51].In : WORD  // In.IoData.IoData[3]
        input  std12k5.AI_K[52].In : WORD  // In.IoData.IoData[4]
        input  std12k5.AI_K[53].In : WORD  // In.IoData.IoData[5]
        input  std12k5.AI_K[54].In : WORD  // In.IoData.IoData[6]
        input  std12k5.AI_K[55].In : WORD  // In.IoData.IoData[7]
        input  std12k5.AI_K[48].Vera : WORD  // Diagnosis.Flags.Veracity
        input  std12k5.MODULES03[16].CH_MODCONF : WORD  // Diagnosis.Service.Service[0]
        input  std12k5.MODULES03[16].CH_ERRNOW : WORD  // Diagnosis.Service.Service[1]
        input  std12k5.MODULES03[16].CH_ERRHIST : WORD  // Diagnosis.Service.Service[2]
        input  std12k5.MODULES03[16].CH_NDIAG : WORD  // Diagnosis.Service.Service[3]
        input  std12k5.MODULES03[16].CH_MDIAG : WORD  // Diagnosis.Service.Service[4]
        input  std12k5.MODULES03[16].CH_FIRMVER : WORD  // Diagnosis.Service.Service[5]
        input  std12k5.MODULES03[16].CH_FIRMDATE : WORD  // Diagnosis.Service.Service[6]
        unmapped channels: In, Diagnosis
  libraries: Standard, * (System); CmpLog, 3.5.2.0 (System); SysFileStream23, 3.5.2.0 (System); SysTypes Interfaces, * (System); Util, * (System); Unit Conversion Interfaces, * (Intern); FloatingPointUtils, * (System); CAA List And Tree, 3.5.0.0 (CAA Technical Workgroup); SysTime, 3.4.1.20 (System); CmpErrors, 3.3.1.40 (System)
  LowLevel_Algoritms/
    algoritms/
      function block Rassoglasovanie_dPmg [ST]
      function block AiProtectionDual [ST]: reset
      function block Krans_Protections [ST]: reset
      function block DiProtection_fb [ST]: reset
      function block DiProtection [ST]: reset
      function block MvProtection [ST]: reset
      function block AiProtection [ST]: reset, run
    Common/
      function block everifingTrue [ST]
      function DisableAiLimits [ST]
      function EnableAiLimits [ST]
      function getLimitFlags [ST]
    im/
      function block IMs [ST]
      function block Krans_Sdvig [ST]
      function block NasosNu [ST]: Off
      function block Krans_Sdvig_kr4 [ST]
      function block Reability [ST]
      function block Kr4 [ST]
  lowLevel_ecl/
    Common/
      function block BaseObject [ST]: FB_init, getNext, setDefaultPersistent, SaveToFile, LoadFromFile, readPersistent, writePersistent, writeValue, readValue, onInit, registerInAcrhive
      fb/
        function block AnalogRecalc [ST]
        function block RP_trig [ST]
        function block RsRTrig [ST]
        function block unpackTime [ST]
      functions/
        function checkArg [ST]
        function HexString_to_Word [ST]
        function rABS [ST]
        function RNaN [ST]
        function validAndTrue [ST]
      parameters/
        AnalogParameter/
          function block AnalogParametr [ST]: processCmd, readPersistent, setValue, writePersistent
          function block AnalogParametrDinamic [ST]: processCmd, setValue
          function block BaseAnalogParametr [ST]: getValue, isValidValue, setValue
          interface IAnalogParameter: setValue
          interface IAnalogValue: getValue
          function block RefToRealAnalogParameter [ST]: getValue
        function block DiscretParametr [ST]: processCmd, readPersistent, setValue, writeImStatus, writePersistent
        question/
          data type Answers
          function block Question [ST]: ask, processCmd, reseiveAnswer, reset, writeImStatus
        function block TimeParametr [ST]: processCmd, readPersistent, setValue, writePersistent
      function block AloneLogMessage [ST]: write
      smartPack/
        function block smartPack [ST]: reset, setBit, setBits
        function block SmartUnpack [ST]: getBit, getBits
        function block smartWordPack [ST]: reset, setBit, setBits
      table/
        function callExec [ST]
        function callObject [ST]
        data type TableDescriptor
    kontroller/
      function ExecKontrollersComands [ST]
      function execKontrollersInputs [ST]
      function execKontrollersOutputs [ST]
      extSources/
        function block AiMovingSverage [ST]: disabledAlarms, GetData, getLast, imit, writeNext
        data type MultiAnalogLimits
        function block TripledAnalog [ST]: GetData, imit, initArray, compare, sort, validateInputs
        data type AnalogItem
        data type AnalogsProcessing
        function block MultiAnalog [ST]: CalkLimits, disabledAlarms, GetData, imit, onInit, CalcLLHl, checkInputs, getNextFirstValid, getNextLastValid, initArray, InputIntervalsCnt, isValidInput, readPersistent, averageValue, maxValue, medianValue, minValue, compare, sort, writePersistent
      mlp/
        Sources/
          function block AoSourceMlp [ST]: setKontroller, writeData
          function block AiFrequenceMlp [ST]: readPersistent, setKontroller, GetData, writePersistent, setDefaultPersistent
          function block DiSourceMlp [ST]: setKontroller, getData
          function block AnalogDiSourceMlp [ST]: readPersistent, writePersistent, setLimits, processCmd, setKontroller
          function block AiSourceMlp [ST]: setKontroller, GetData
          function block DoSourceMlp [ST]: setKontroller, writeData
          interface IMlpSource: setKontroller
        data type sDIN_DOUT
        global variables FAUs
        data type AIn_s
        data type DIn_s
        data type sAIN_AOUT
        data type TypeUSO
        data type DiagnosticIndex
        Diagnostic/
          function block DiagnosticMlp [ST]: WriteConfig, writeStatus, ReadModules, FaultModel, readDi8Status, readAI4Status, readOA4Status, readConfig, readConfig_faleev
          iniFile/
            function block iniFileReader [ST]: open, close, readLn
            data type iniFileLine
            data type iniFileStatus
          data type BsDescriptor
          data type ModuleDescriptor
          data type BsStatusDecriptor
          data type ModuleStatusDescriptor
          data type ModuleTypes
        function block Elpk04 [ST]: callSetController
      baseSources/
        function block DISource [ST]: archName, archReliability, archValue, getData, imit
        function block DOSource [ST]: archName, archReliability, archValue, imit, setValue, writeData
        interface IAiSource: aiInterval, aiRemont, aiValue
        function block InversableReliableBit [ST]: inverse, setReliability, setValue
        interface ISource: imit
        function block ReliableBit [ST]: ReliableFalse, ReliableTrue, setReliability, setValue
        data type statusAi
        function block AISource [ST]: aiInterval, aiRemont, aiValue, apFilter, archName, archSrcValue, archStatus, archValue, CalkLimits, disabledAlarms, exponential, GetData, imit, kvitNotReliable, notReliable, processCmd, readPersistent, resetRemont, setDefaultPersistent, setRemont, setUstavki, writeImStatus, writePersistent
        data type AnalogAlarms
        data type AnalogLimitFlags
        function block AOSource [ST]: archSrcValue, archValue, cmdSetValue, imit, processCmd, readPersistent, setDefaultPersistent, setLimits, setValue, writeData, writePersistent
        function block CustomSource [ST]: imit
      function block baseKontroller [ST]: callOutputTable, setImit, callCommands, callInputTable
      interface IKontroller: callCommands, callInputTable, callOutputTable
      modbus/
        data type MbAiWordOrder
        function block MbKontroller [ST]: callInputTable, callOutputTable, getInputFloat, getInputValue, ProcessInputs, ProcessOutputs, setOutputByte, setOutputFloat, setOutputValue, setSourcesProp
        data type MbKontrollerRole
        function block MlpMbKontroller [ST]: getInputFloat, getInputValue, setOutputByte, setOutputFloat, setOutputValue
        Sources/
          function block AiSourceMb [ST]: GetData, setKontroller
          function block AoProxiMb [ST]: setKontroller, writeData
          function block DiSourceMb [ST]: getData, setKontroller
          function block DoSourceMb [ST]: setKontroller, writeData
          data type FloatAsWords
          interface IMbSource: setKontroller
          SpecSources/
            function block AiSourceMbByte [ST]: GetData
            function block AiSourceMbWord [ST]: GetData
            function block AoProxiMbByte [ST]: writeData
            function block AoProxiMbWord [ST]: writeData
        data type UsedByteMBSource
    im/
      BaseIms/
        function block BaseIm [ST]: archName, archStatus, DisableOpcControl, EnableOpcControl, execCommand, hasCommand, opcCommandsDisabled, writeCommandToStatus, processObjectTable, checkCmd, resetCommand, errorCommand, onCommandActive, processCmd, setCmd, sendCommand, writeImStatus, CommandFail
        data type cmdSources
        function block DualStateIm [ST]: off, calcStatus, getSdvig, getStatus, onInit, resetCommand, noStatusLinks, resetOuts, on, writeImStatus
        function block DualStateKran [ST]: close, off, reset, on, open, doOpenCloseCmd, onCommandActive, processCmd, resetCommand
        function block DualStateSwitch [ST]: on, resetOutputs, onCommandActive, processCmd, resetCommand, off
        interface ObjectCommands: DisableOpcControl, execCommand, hasCommand, EnableOpcControl, writeImStatus
        function block singleSignal [ST]: writeImStatus
        data type statusDualInput
        function block singleOutput [ST]: on, processCmd, impulse, off
      extensions/
        function block ExtNarabotka [ST]: readPersistent, reset, start, started, stop, writePersistent
      Kran/
        function block Kran [ST]: getSdvig, writeImStatus
      Mokveld/
        function block Mokveld [ST]: calcOnStatus, cmdSetTarget, processCmd, readPersistent, setDefaultPersistent, setTarget, writeImStatus, writePersistent
      sectionSwitch/
        data type basketStats
        function block SectionSwitch [ST]: on, processCmd, resetPlakat, setPlakat, writeImStatus
      ventvs/
        function block Nasos [ST]
        function block Switch [ST]
        function block Ten [ST]
        function block Vent [ST]
        function block Ventvs [ST]: lastComandIsOn, getSdvig, writeImStatus
        function block Zaslonka [ST]
      Zadvigka/
        function block Zadvigka [ST]: getSdvig, writeImStatus
    EmergencyAarchive/
      function block Archive [ST]: appendSource, newTimeSlice, lastTimeSlice, firstTimeSlice, timeToString, timeTofileName, uintToStrf, writeHead, writeDataRow, countinueDataWrite, register, FB_init, startAccident, writeLog
      function block TimeSlice [ST]: appendValueListener, copy, update, timeStamp, FB_Exit
      function block ArchiveProvider [ST]: RegisterArchive, RegisterSource, accidentStarted
      ObjectListener/
        function createObjectListener [ST]
        function block ImObjectListener [ST]: copy, getName, update, getParametersCount, getParametrValue, getParametrName
        interface IImArchObject: archStatus
        function block AnalogObjectListener [ST]: copy, getName, update, getParametersCount, getParametrName, getParametrValue
        interface IBaseArchObject: archName
        interface IAnalogArchObject: archValue, archSrcValue
        interface IDiscretArchObject: archValue, archReliability
        function block DiscretObjectListener [ST]: copy, getName, update, getParametersCount, getParametrName, getParametrValue
        interface IObjectListener: copy, getName, update, getParametersCount, getParametrName, getParametrValue
        function deleteObjectListener [ST]
    algoritms/
      interface AlgoritmInterface: autoRun, callBase, CanRun, isRuning, reset, run
      function block BaseAlgoritm [ST]: autoRun, callBase, CanRun, end, getTable, hasError, isEnded, isRuning, onInit, processCmd, processObjectTable, reset, run, writeImStatus
      function block BaseAlgoritmsManager [ST]: onInit, onStart, processCmd
      function block BaseProtection [ST]: check, processCmd, readPersistent, remont, reset, resetRemont, run, setRemont, signaling, writeImStatus, writePersistent
      function ExecComands [ST]
      interface IProtection: check, remont, signaling
      phases/
        data type DualStateImAction
        interface IAlgoritmPhase: error, getPhaseNum, reset, run, setBlockIm, start, top
        function block ph_algoritm [ST]: getError, GetIm, getTop, onRun
        function block ph_Analog [ST]: getError, GetIm, getTop, onRun
        function block ph_Kran [ST]: getError, GetIm, getTop, onRun
        function block ph_SingleOutput [ST]: getError, GetIm, getTop, onRun
        function block ph_SingleSignal [ST]: getError, GetIm, getTop
        function block ph_Switch [ST]: getError, GetIm, getTop, onRun
        function block ph_Timer [ST]: getDelay, getTop, onReset, onRun
        function block ph_WaitAnalogValue [ST]: getError, GetIm, getTop, onRun
        function block BaseAlgoritmPhase [ST]: error, getError, GetIm, getPhaseNum, getTop, onReset, onRun, reset, run, setBlockIm, start, top
        function block CustomPhase [ST]: getPhaseNum, onReset, onRun, reset, run, setBlockIm, start, top, error
        data type PhaseAlgoritmAction
      function runAlg [ST]
      function block StepBySteapAlgoritm [ST]: allPhasesDone, hasError, ProcessPhases, reset, run, writeImStatus
  text list GlobalTextList
  REZERV1/
    function ADDCRC16 [ST]
    function block COM_Rd [ST]
    function block COM_Wr [ST]
    function block COM1 [ST]
    function block PilaReady [ST]
    function block PilaStat [ST]
    function block PilaTst [ST]
    function block REZ1 [ST]
    function block REZ2_1 [ST]
    data type RezervState
    function block SetStateK [ST]
    function ADDCRC16_1 [ST]
    program REZERV1 [ST]
    program REZERV2 [ST]
  Elpk_03_02_COMMON/
    program ELPK03_to_MLP_IN [ST]
    program ELPK03_to_MLP_OUT [ST]
    data type T_DI03
    data type T_AI03
    data type T_DIAGNOSTIC03
    function AI_03_RR [ST]
    function DI_03_R [ST]
    data type T_DO03
    function DO_03_kk [ST]
*)

// K1/std12k5/hardwareConfig/AOConfig
TYPE AOConfig:
	STRUCT
		//AoName:AoSourceMlp(table:=ADR(kontroller.outputTable)):=(addr:=0);
	END_STRUCT
END_TYPE

// K1/std12k5/hardwareConfig/DOConfig
TYPE DOConfig:
	STRUCT
		do_0:DoSourceMlp(table:=ADR(kontroller.outputTable)):=(addr:=0);
		do_1:DoSourceMlp(table:=ADR(kontroller.outputTable)):=(addr:=1);
		do_2:DoSourceMlp(table:=ADR(kontroller.outputTable)):=(addr:=2);
		do_3:DoSourceMlp(table:=ADR(kontroller.outputTable)):=(addr:=3);
		do_4:DoSourceMlp(table:=ADR(kontroller.outputTable)):=(addr:=4);	
	END_STRUCT
END_TYPE

// K1/std12k5/algoritms/AlgoritmsConfig
TYPE AlgoritmsConfig:
		{attribute 'symbol' := 'read'}
	STRUCT
		opcComands:OpcCommands(table:=algManager.getTable());
		Auto_Avom_:AutoAVOM (table:=algManager.getTable()):=(T_posle_AVOM:=ai.TMaslaPosleAVOM, A1:=im.v1_Avom, A2:=im.v2_Avom, A3:=im.v3_Avom, A4:=im.v4_Avom);
		autoNu_1:AutoNuAlg_1(table:=algManager.getTable()):=(nu:=Im.nu,di:=im.PerepadDavlenieMasloGaz_Less100, di_CK:=im.PerepadDavlenieMasloGaz_CK);
		autoNu_2:AutoNuAlg_2(table:=algManager.getTable()):=(nu:=Im.nu,di:=im.PerepadDavlenieMasloGaz_Less100, di_CK:=im.PerepadDavlenieMasloGaz_CK);
		autoPns:AutoPnsAlg(table:=algManager.getTable()):=(pns:=Im.pns,Psm_GNS:=ai.DavlenijaMaslaPosleGNS);
		AUto_Ten_:AutoTEn (table:=algManager.getTable()):=(Tmb:=ai.TMaslaMB, TmbTEN:=ai.TMaslaMB_TEN, TEN:=im.TEN_MB, CMN:=im.CMN);
		PNS_ON_MV_:PNS_ON_MV_ON (table:=algManager.getTable()):=(PNS:=im.PNS);
		no:noAlg(table:=algManager.getTable()):=(BlockIm:=FALSE);
		ao:aoAlg(table:=algManager.getTable()):=(BlockIm:=FALSE);
		Opres:Opressovka (table:=algManager.getTable()):=(BlockIm:=FALSE);
		Pms:Prov_Pms (table:=algManager.getTable()):=(BlockIm:=FALSE);
		dPmg:Prov_dPmg (table:=algManager.getTable()):=(BlockIm:=FALSE);
		ppu:ppuAlg(table:=algManager.getTable());
		F1_1:puskFirst_faza1 (table:=algManager.getTable()):=(BlockIm:=FALSE);
		F1_2:puskFirst_faza2 (table:=algManager.getTable()):=(BlockIm:=FALSE);
		F2_Ch:puskSecond_faza_Chastotny (table:=algManager.getTable()):=(BlockIm:=FALSE);
		F2_R:puskSecond_faza_Reactor (table:=algManager.getTable()):=(BlockIm:=FALSE);
		F3:puskThird_faza (table:=algManager.getTable()):=(BlockIm:=FALSE);
		F4:Kran_6_Close (table:=algManager.getTable()):=(BlockIm:=FALSE);
		Kr6_Move: Kran_6_Move (table:=algManager.getTable()):=(BlockIm:=FALSE);
		AutoPNS_Start:PNS_Pusk (table:=algManager.getTable()):=(BlockIm:=FALSE);
		R_AutoAVom:Reset_AutoAVOM (table:=algManager.getTable()):=(BlockIm:=FALSE);
		R_AutoTEN:Reset_AutoTEN (table:=algManager.getTable()):=(BlockIm:=FALSE);
		R_TestIM:Reset_Test_IM (table:=algManager.getTable()):=(BlockIm:=FALSE);
		S_AutoAVOM: Start_AutoAVOM (table:=algManager.getTable()):=(BlockIm:=FALSE);
		S_AutoTEN: Start_AutoTEN (table:=algManager.getTable()):=(BlockIm:=FALSE);
		S_Test_IM: Start_Test_IM (table:=algManager.getTable()):=(BlockIm:=FALSE);
		S_Vibr: Start_ProtectionsVibr(table:=algManager.getTable()):=(BlockIm:=FALSE);
		S_dPmg: Start_Prov_dPmg (table:=algManager.getTable()):=(BlockIm:=FALSE);
		S_I:	Start_Prov_I (table:=algManager.getTable()):=(BlockIm:=FALSE);
		S_K:	Start_Prov_k (table:=algManager.getTable()):=(BlockIm:=FALSE);
		S_Pms:	Start_Prov_Pms (table:=algManager.getTable()):=(BlockIm:=FALSE);
		S_V:	Start_Prov_V (table:=algManager.getTable()):=(BlockIm:=FALSE);
		S_AP:	Start_Pusk_AP (table:=algManager.getTable()):=(BlockIm:=FALSE);
		S_PP:	Start_Pusk_PP (table:=algManager.getTable()):=(BlockIm:=FALSE);
		S_NO:	Start_NO (table:=algManager.getTable()):=(BlockIm:=FALSE);
		S_AO:	Start_AO (table:=algManager.getTable()):=(BlockIm:=FALSE);
		Test_IM: TestIMAlg (table:=algManager.getTable());
		Synch_Rejim_:Synch_Rejims (table:=algManager.getTable());
		Kran4_Samosdvig:Krans_Sdvig_kr4(table:=algManager.getTable()):=(Krans:=im.kran4, block:=ystavki.blockkr4, block_from_alg:=ystavki.Block_kr4_alg);
		Kran1_Samosdvig:Krans_Sdvig_kr4(table:=algManager.getTable()):=(Krans:=im.kran1, block:=ystavki.blockkr1, block_from_alg:=ystavki.Block_kr1_alg); 
		Kran2_Samosdvig:Krans_Sdvig_kr4(table:=algManager.getTable()):=(Krans:=im.kran2, block:=ystavki.blockkr2, block_from_alg:=ystavki.Block_kr2_alg);
		Kran3_Samosdvig:Krans_Sdvig_kr4(table:=algManager.getTable()):=(Krans:=im.kran3, block:=ystavki.blockkr3, block_from_alg:=ystavki.Block_kr3_alg);
		Kran3b_Samosdvig:Krans_Sdvig_kr4(table:=algManager.getTable()):=(Krans:=im.kran3b, block:=ystavki.blockkr3b, block_from_alg:=ystavki.Block_kr3b_alg);
		
		Kran5_Samosdvig:Krans_Sdvig_kr4(table:=algManager.getTable()):=(Krans:=im.kran5, block:=ystavki.blockkr5, block_from_alg:=ystavki.Block_kr5_alg);
		Kran6_Samosdvig:Krans_Sdvig_kr4(table:=algManager.getTable()):=(Krans:=im.kran6, block:=ystavki.blockkr6, block_from_alg:=ystavki.Block_kr6_alg);
		
		Test_P:Test_Protections (table:=algManager.getTable()):=();
		Start_Test_P:Start_Test_Pr (table:=algManager.getTable()):=();
		
	END_STRUCT
END_TYPE

// K1/std12k5/hardwareConfig/AiConfig
TYPE AiConfig:
	STRUCT
		///////////////////////////////////////////////////////////////////////////////////////////////////////////////
		//{name:Температура стали статора 1 канал}
		TStalisStatoraKanall:AI_Final(table:=ADR(kontroller.inputTable)):=(addr:=0, dLL:=0,dHL:=150, dHW:=130, histeresis:=0.5);
		//{name:Температура стали статора 2 канал}
		TStalisStatoraKanal2:AI_Final(table:=ADR(kontroller.inputTable)):=(addr:=1, dLL:=0,dHL:=150, dHW:=130, histeresis:=0.5);
		//{name:Температура стали статора 3 канал}
		TStalisStatoraKanal3:AI_Final(table:=ADR(kontroller.inputTable)):=(addr:=2, dLL:=0,dHL:=150, dHW:=130, histeresis:=0.5);
	
		///////////////////////////////////////////////////////////////////////////////////////////////////////////////
		//{name:Температура меди статора 1 канал}
		TMediStatoraKanall:AI_Final(table:=ADR(kontroller.inputTable)):=(addr:=3, dLL:=0,dHL:=150, dHW:=130, histeresis:=0.5);
		//{name:Температура меди статора 2 канал}
		TMediStatoraKanal2:AI_Final(table:=ADR(kontroller.inputTable)):=(addr:=4, dLL:=0,dHL:=150, dHW:=130, histeresis:=0.5);
		//{name:Температура меди статора 3 канал}
		TMediStatoraKanal3:AI_Final(table:=ADR(kontroller.inputTable)):=(addr:=5, dLL:=0,dHL:=150, dHW:=130, histeresis:=0.5);
		
		
	
		
		///////////////////////////////////////////////////////////////////////////////////////////////////////////////
		//{name:Температура опорного подшипника ЭД т.1 }
		TOpornogoPodshipnikaEDT_1:AI_Final_SIP(table:=ADR(kontroller.inputTable)):=(addr:=6, dLL:=0,dHL:=100,dHW:=75,dHA:=80,  histeresis:=0.5, ChangeSIP:=(value:=10));
		//{name:Температура опорно-упорного подшипника ЭД т.2}
		TOpornoYpornogoPodshipnikaEDT_2:AI_Final_SIP(table:=ADR(kontroller.inputTable)):=(addr:=7,dLL:=0,dHL:=100,dHW:=75,dHA:=80, histeresis:=0.5, ChangeSIP:=(value:=10));
		//{name:Температура опорно-упорного подшипника колеса редуктора со стороны ЭД т.3}
		TOpornoYpornogoPodshipnikaKolesaRedEDT_3:AI_Final_SIP(table:=ADR(kontroller.inputTable)):=(addr:=8, dLL:=0,dHL:=100,dHW:=75,dHA:=80,  histeresis:=0.5, ChangeSIP:=(value:=10));
		//{name:Температура опорно-упорного подшипника колеса редуктора со стороны Нагнетателя т.4}
		TOpornoYpornogoPodshipnikaKolesaRedHT_4:AI_Final_SIP(table:=ADR(kontroller.inputTable)):=(addr:=9, dLL:=0,dHL:=100,dHW:=75,dHA:=80,   histeresis:=0.5, ChangeSIP:=(value:=10));
		//{name:Температура опорного подшипника шестерни редуктора со стороны ЭД т.5 }
		TOpornogoPodshipnikaShesterniReduktoraT_5:AI_Final_SIP(table:=ADR(kontroller.inputTable)):=(addr:=10, dLL:=0,dHL:=100,dHW:=75,dHA:=80,   histeresis:=0.5, ChangeSIP:=(value:=10));
		//{name:Температура опорного подшипника редуктора со стороны Нагнетателя т.6}
		TOpornogoPodshipnikaReduktoraHT_6:AI_Final_SIP(table:=ADR(kontroller.inputTable)):=(addr:=11, dLL:=0,dHL:=100,dHW:=75,dHA:=80,  histeresis:=0.5, ChangeSIP:=(value:=10));
		//{name:Температура опорно-упорного подшипника нагнетателя т.7.1}
		TOpornoYpornogoPodshipnikaNagnetateljaT_7_1:AI_Final_SIP(table:=ADR(kontroller.inputTable)):=(addr:=12, dLL:=0,dHL:=100,dHW:=75,dHA:=80,   histeresis:=0.5, ChangeSIP:=(value:=10));
		//{name:Температура опорно-упорного подшипника нагнетателя т.7.2}
		TOpornoYpornogoPodshipnikaNagnetateljaT_7_2:AI_Final_SIP(table:=ADR(kontroller.inputTable)):=(addr:=13, dLL:=0,dHL:=100,dHW:=75,dHA:=80,  histeresis:=0.5, ChangeSIP:=(value:=10));
		//{name:Температура опорно-упорного подшипника свободного конца нагнетателя т.8.1}
		TOpornoYpornogoPodshipnikaSvobodnogoKoncaNT_8_1:AI_Final_SIP(table:=ADR(kontroller.inputTable)):=(addr:=14, dLL:=0,dHL:=100,dHW:=75,dHA:=80,   histeresis:=0.5, ChangeSIP:=(value:=10));
		//{name:Температура порно-упорного подшипника свободного конца нагнетателя т.8.2}
		TOpornoYpornogoPodshipnikaSvobodnogoKoncaNT_8_2:AI_Final_SIP(table:=ADR(kontroller.inputTable)):=(addr:=15, dLL:=0,dHL:=100,dHW:=75,dHA:=80,   histeresis:=0.5, ChangeSIP:=(value:=10));
		//{name:Температура упорного подшибника рабочих колодок нагнетателя т.9.1}
		TYpornogoPodshipnikaRavKolodokHT_9_1:AI_Final_SIP(table:=ADR(kontroller.inputTable)):=(addr:=16, dLL:=0,dHL:=100,dHW:=75,dHA:=80,   histeresis:=0.5, ChangeSIP:=(value:=10));
		//{name:Температура упорного подшибника рабочих колодок нагнетателя т.9.2}
		TYpornogoPodshipnikaRavKolodokHT_9_2:AI_Final_SIP(table:=ADR(kontroller.inputTable)):=(addr:=17, dLL:=0,dHL:=100,dHW:=75,dHA:=80,   histeresis:=0.5, ChangeSIP:=(value:=10));
		//{name:Температура нерабочих колодок упорного подшипника нагнетателя т.10.1}
		TYpornogoPodshipnikaNerabKolodokHT_10_1:AI_Final_SIP(table:=ADR(kontroller.inputTable)):=(addr:=18, dLL:=0,dHL:=100,dHW:=75,dHA:=80,   histeresis:=0.5, ChangeSIP:=(value:=10));
		//{name:Температура нерабочих колодок упорного подшипника нагнетателя т.10.2}
		TYpornogoPodshipnikaNerabKolodokHT_10_2:AI_Final_SIP(table:=ADR(kontroller.inputTable)):=(addr:=19, dLL:=0,dHL:=100,dHW:=75,dHA:=80,   histeresis:=0.5, ChangeSIP:=(value:=10));
		///////////////////////////////////////////////////////////////////////////////////////////////////////////////
		//{name:Температура холодного воздуха ЭД 1 канал}
		THolodnogoVozduhaEDKanall:AI_Final(table:=ADR(kontroller.inputTable)):=(addr:=20, dLL:=0,dHL:=100, dHW:=60, histeresis:=0.5);
		//{name:Температура холодного воздуха ЭД 2 канал}
		THolodnogoVozduhaEDKanal2:AI_Final(table:=ADR(kontroller.inputTable)):=(addr:=21, dLL:=0,dHL:=100, dHW:=60, histeresis:=0.5);
		
			///////////////////////////////////////////////////////////////////////////////////////////////////////////////
		//{name:Температура горячего воздуха ЭД 1 канал}
		TGorjachegoVozduhaEDKanall:AI_Final(table:=ADR(kontroller.inputTable)):=(addr:=22, dLL:= 0,dHL:=100, dHW:=70, histeresis:=0.5);
		//{name:Температура горячего воздуха ЭД 2 канал}
		TGorjachegoVozduhaEDKanal2:AI_Final(table:=ADR(kontroller.inputTable)):=(addr:=23, dLL:= 0,dHL:=100, dHW:=70, histeresis:=0.5);
		
		//{name:Температура Наружного воздуха}
		TNArujnogoVozduha:AI_Final(table:=ADR(kontroller.inputTable)):=(addr:=24, dLL:=-50,dHL:=100, histeresis:=0.5);
		
		
		
		///////////////////////////////////////////////////////////////////////////////////////////////////////////////
		//{name:Температура газа на входе нагнетателя}
		TgazaNaVhodeH:AI_Final(table:=ADR(kontroller.inputTable)):=(addr:=25, dLL:=-50,dHL:=100,dHW:=80, histeresis:=0.5);
		//{name:Температура газа на выходе нагнетателя}
		TgazaNaVyhodeH:AI_Final_SIP(table:=ADR(kontroller.inputTable)):=(addr:=26, dLL:=-50,dHL:=100,dHW:=80,dHA:=90,   histeresis:=0.5, ChangeSIP:=(value:=10));
		
		///////////////////////////////////////////////////////////////////////////////////////////////////////////////
		//{name:Температура масла до АВОМ}
		TMasladoAVOM:AI_Final(table:=ADR(kontroller.inputTable)):=(addr:=27, dLL:=0,dHL:=150,dHW:=55, histeresis:=0.5);
		//{name:Температура масла после АВОМ}
		TMaslaPosleAVOM:AI_Final_SIP(table:=ADR(kontroller.inputTable)):=(addr:=28, dLL:=0,dHL:=150,dHW:=55,   histeresis:=0.5, ChangeSIP:=(value:=10));
		
		///////////////////////////////////////////////////////////////////////////////////////////////////////////////
		//{name:Температура масла в маслобаке}
		TMaslaMB:AI_Final_SIP(table:=ADR(kontroller.inputTable)):=(addr:=29, dLL:=0,dHL:=150,dLW:=25,   histeresis:=0.5, ChangeSIP:=(value:=10));
		//{name:Температура масла в маслобаке над ТЭН}
		TMaslaMB_TEN:AI_Final_SIP(table:=ADR(kontroller.inputTable)):=(addr:=30, dLL:=0,dHL:=100,dHW:=50,  histeresis:=0.5, ChangeSIP:=(value:=10));
		//{name:Температура в ШУ}
		TEmperatura_v_SHU:AI_Final(table:=ADR(kontroller.inputTable)):=(addr:=32, dLL:=-40,dHL:=100, rassoglasovanie:=2, histeresis:=0.5);
		
		///////////////////////////////////////////////////////////////////////////////////////////////////////////////
		//{name:Давление масла смазки низкое }
		DavlenijaMasloSmNizkoe:AI_Final(table:=ADR(kontroller.inputTable)):=(addr:=33, dLL:=0,dHL:=400,dLW:=50, dLA:=25, rassoglasovanie:=1.5, histeresis:=0.5);
		//{name:Перепад давления масла на масляном фильтре}
		PerepadDavlenieNaMasloFiltre:AI_Final(table:=ADR(kontroller.inputTable)):=(addr:=34, dLL:=0,dHL:=250,dHW:=150, rassoglasovanie:=1.5, histeresis:=0.5);	
		//{name:Давление масла смазки высокое}
		DavlenijaMasloSmVysokoe:AI_Final(table:=ADR(kontroller.inputTable)):=(addr:=35, dLL:=0,dHL:=1000,dLW:=300, dLA:=250, rassoglasovanie:=1.5, histeresis:=0.5);
		//{name:Давление масла смазки после ГНС }
		DavlenijaMaslaPosleGNS:AI_Final(table:=ADR(kontroller.inputTable)):=(addr:=36, dLL:=0,dHL:=1000,dLW:=450, rassoglasovanie:=1.5, histeresis:=0.5);
		//{name:Давление масла после Насоса уплотнения }
		DavlenijaMaslaPosleNU:AI_Final(table:=ADR(kontroller.inputTable)):=(addr:=37, dLL:=0,dHL:=10, dLW:=3, rassoglasovanie:=1.5, histeresis:=0.5);
		///////////////////////////////////////////////////////////////////////////////////////////////////////////////
		
		//{name:Перепад давления газа на Конфузоре}
		PerepadDavlenieNaKonfuzore:AI_Final(table:=ADR(kontroller.inputTable)):=(addr:=40, dLL:=0,dHL:=250, dLW:=15, rassoglasovanie:=1.5, histeresis:=0.5);
		
		/////////////////////////////////////////////////////////////////////////////////////////////////////////////// 
		//{name:Осевой сдвиг нагнетателя +}
		OsSdvigNagnetatelja_Plus:AI_Final(table:=ADR(kontroller.inputTable)):=(addr:=42, dLL:=0,dHL:=1000,dHW:=200, dHA:=300, rassoglasovanie:=1.5, histeresis:=0.5);
		//{name:Осевой сдвиг нагнетателя -}
		OsSdvigNagnetatelja_Minus:AI_Final(table:=ADR(kontroller.inputTable)):=(addr:=43, dLL:=0,dHL:=1000,dHW:=200, dHA:=300, rassoglasovanie:=1.5, histeresis:=0.5); 
		/////////////////////////////////////////////////////////////////////////////////////////////////////////////// 
		//{name:Перепад давления масло-газ }
		PerepadDavlenieMasloGaz:AI_Final(table:=ADR(kontroller.inputTable)):=(addr:=41, dLL:=0,dHL:=1600,dLW:=150, dLA:=100, rassoglasovanie:=1.5);
		///////////////////////////////////////////////////////////////////////////////////////////////////////////////
		//{name:Давление газа на входе нагне-тателя }
		DGazaNaVhodeNagnetatelja:AI_Final(table:=ADR(kontroller.inputTable)):=(addr:=44, dLL:=0,dHL:=10, dLW:=4.895(*, dLA:=4.589*), rassoglasovanie:=1.5, histeresis:=0.5);
		//{name:Давление газа на выходе нагне-тателя }
		DGazaNaVyhodeNagnetatelja:AI_Final(table:=ADR(kontroller.inputTable)):=(addr:=45, dLL:=0, dHL:=10, dHW:=7.55, dHA:=7.653, rassoglasovanie:=1.5, histeresis:=0.5);
		//{name: Давление импульсного газа}
		DavlenieImpulsGaz:AI_Final(table:=ADR(kontroller.inputTable)):=(addr:=46, dLL:=0, dHL:=10, dLW:=5, rassoglasovanie:=1.5, histeresis:=0.5);
		//{name: Уровень масла в маслобаке}
		YrovenMaslaMB:AI_Final(table:=ADR(kontroller.inputTable)):=(addr:=48, dLL:=190,dHL:=885, dLW:=530, rassoglasovanie:=1.5, histeresis:=0.5);
		
		///////////////////////////////////////////////////////////////////////////////////////////////////////////////
		//{name:Контроль ~220В}
		Kontrol_per220V:AI_Final(table:=ADR(kontroller.inputTable)):=(addr:=52, dLL:=0,dHL:=250,dLW:=187,dHW:=242, rassoglasovanie:=1.5, histeresis:=0.5);
		//{name:Контроль =220В}
		Kontrol_post220V:AI_Final(table:=ADR(kontroller.inputTable)):=(addr:=53, dLL:=0,dHL:=250,dLW:=187,dHW:=242, rassoglasovanie:=1.5, histeresis:=0.5);
		
		///////////////////////////////////////////////////////////////////////////////////////////////////////////////
		//{name:Виброскорость опорного подшипника ЭД т.1 }
		VibroSkorostOPED_T1:AI_Final(table:=ADR(kontroller.inputTable)):=(addr:=56, dLL:=0,dHL:=25,dHW:=11, dHA:=18, rassoglasovanie:=1.5, histeresis:=0.5);
		//{name:Виброскорость опорно-упорного подшипника ЭД со стороны редуктора т.2 }
		VibroSkorostOYPED_T2:AI_Final(table:=ADR(kontroller.inputTable)):=(addr:=57, dLL:=0,dHL:=25,dHW:=11, dHA:=18, rassoglasovanie:=1.5, histeresis:=0.5);
		//{name:Виброскорость опорно-упорного подшипника колеса редуктора со стороны ЭД т.3 }
		VibroSkorostOYPKolesaED_T3:AI_Final(table:=ADR(kontroller.inputTable)):=(addr:=58, dLL:=0,dHL:=25,dHW:=11, dHA:=18, rassoglasovanie:=1.5, histeresis:=0.5);
		//{name:Виброскорость опорного подшипника колеса редуктора со стороны нагнетателя т.4 }
		VibroSkorostOPKolesaRH_T4:AI_Final(table:=ADR(kontroller.inputTable)):=(addr:=59, dLL:=0,dHL:=25,dHW:=11, dHA:=18, rassoglasovanie:=1.5, histeresis:=0.5);
		//{name:Виброскорость опорного подшипника шестерни редуктора со стороны ЭД т.5 }
		VibroSkorostOPShesterniRED_T5:AI_Final(table:=ADR(kontroller.inputTable)):=(addr:=60, dLL:=0,dHL:=25,dHW:=11, dHA:=18, rassoglasovanie:=1.5, histeresis:=0.5);
		//{name:Виброскорость опорного подшипника шестерни редуктора со стороны нагнететеля т.6}
		VibroSkorostOPShesterniReduktoraH_T6:AI_Final(table:=ADR(kontroller.inputTable)):=(addr:=61, dLL:=0,dHL:=25,dHW:=11, dHA:=18, rassoglasovanie:=1.5, histeresis:=0.5);
		
		
		
		//{name:Ток статора}
		TokStatora:AI_Final(table:=ADR(kontroller.inputTable)):=(addr:=65, dLL:=0,dHL:=1000,dLW:=300, rassoglasovanie:=1.5, histeresis:=0.5);
		
		
		
		
		///////////////////////////////////////////////////////////////////////////////////////////////////////////////	
	END_STRUCT
END_TYPE

// K1/std12k5/algoritms/ImConfig
TYPE ImConfig:
	{attribute 'symbol' := 'readwrite'}
	STRUCT
		//u1:singleSignal(table:=ADR(imTable)):=(signal:=di.di_0.bits[0]);
		/////////***КРАНЫ***///////////////////////////////////////////////////////////////
		///////////////////////////////////////////////////////////////////////////////////
		//{name:Кран 1}	
		kran1:Kran(table:=ADR(imTable)):=(
			statOn:=	di.di_20.bits[5].inverse,
			statOff:=	di.di_20.bits[4].inverse,		
			
			cmdOn:=		od.do_0.bits[0],
			cmdOff:=	od.do_0.bits[1],
			
			inSO:=		di.di_16.bits[0].inverse,
			inSZ:=		di.di_16.bits[1].inverse
		);
		///////////////////////////////////////////////////////////////////////////////////
		//{name:Кран 2}	
		kran2:Kran(table:=ADR(imTable)):=(
			statOn:=	di.di_21.bits[0].inverse,
			statOff:=	di.di_20.bits[7].inverse,
			
			cmdOn:=		od.do_0.bits[2],
			cmdOff:=	od.do_0.bits[3], 
			
			inSO:=		di.di_16.bits[2].inverse,
			inSZ:=		di.di_16.bits[3].inverse
			
		);
		///////////////////////////////////////////////////////////////////////////////////
		//{name:Кран 3}	
		kran3:Kran(table:=ADR(imTable)):=(
			statOn:=	di.di_0.bits[5].inverse,
			statOff:=	di.di_0.bits[4].inverse,
			
			cmdOn:=		od.do_0.bits[4],
			cmdOff:=	od.do_0.bits[5],
			
			inSO:=		di.di_16.bits[4].inverse,
			inSZ:=		di.di_16.bits[5].inverse
		);
		///////////////////////////////////////////////////////////////////////////////////
		//{name:Кран 3'}	
		kran3b:Kran(table:=ADR(imTable)):=(
			statOn:=	di.di_0.bits[7].inverse,
			statOff:=	di.di_0.bits[6].inverse,
			
			cmdOn:=		od.do_0.bits[6],
			cmdOff:=	od.do_0.bits[7],
			
			inSO:=		di.di_16.bits[6].inverse,
			inSZ:=		di.di_16.bits[7].inverse
		);	
		///////////////////////////////////////////////////////////////////////////////////
		//{name:Кран 4}	
		kran4:Kr4(table:=ADR(imTable)):=(
			statOn:=	di.di_1.bits[1].inverse,
			statOff:=	di.di_1.bits[0].inverse,
			
			cmdOn:=		od.do_0.bits[8],
			cmdOff:=	od.do_0.bits[9],
			
			inSO:=		di.di_17.bits[0].inverse,
			inSZ:=		di.di_17.bits[1].inverse
		);	
		///////////////////////////////////////////////////////////////////////////////////
		//{name:Кран 5}	
		kran5:Kran(table:=ADR(imTable)):=(
			statOn:=	di.di_1.bits[3].inverse,
			statOff:=	di.di_1.bits[2].inverse,
			
			cmdOn:=		od.do_0.bits[10],
			cmdOff:=	od.do_0.bits[11],
			
			inSO:=		di.di_17.bits[2].inverse,
			inSZ:=		di.di_17.bits[3].inverse
		);	

		///////////////////////////////////////////////////////////////////////////////////
		//{name:Кран 6}	
		kran6:Kran(table:=ADR(imTable)):=(
			statOn:=	di.di_1.bits[5].inverse,
			statOff:=	di.di_1.bits[4].inverse,		
			
			cmdOn:=		od.do_0.bits[12],
			cmdOff:=	od.do_0.bits[13],
			
			inSO:=		di.di_17.bits[4].inverse,
			inSZ:=		di.di_17.bits[5].inverse
		);
		
		
		
		/////////***ИМ***//////////////////////////////////////////////////////////////////
		///////////////////////////////////////////////////////////////////////////////////
		//{name:МВ}	
		mv: SectionSwitch (table:=ADR(imTable)):=(
			statOn:=	di.di_7.bits[0],
			statOff:=	di.di_20.bits[3],
			
			basketRolledIn:= di.di_7.bits[2].inverse,
			basketRolledOut:= di.di_7.bits[2],
			
			cmdOn:=		od.do_4.bits[6],
			cmdOff:=	od.do_4.bits[7]
		);
		///////////////////////////////////////////////////////////////////////////////////
		//{name:В1 АВОМ}	
		v1_Avom:Avom1(table:=ADR(imTable)):=(
			statOn:=	di.di_5.bits[3],
			statOff:=	di.di_5.bits[3]._inversed,
			
			cmdOn:=		od.do_1.bits[8],
			cmdOff:=	od.do_1.bits[9]
		);		
		///////////////////////////////////////////////////////////////////////////////////
		//{name:В2 АВОМ}	
		v2_Avom:Avom2(table:=ADR(imTable)):=(
			statOn:=	di.di_5.bits[4],
			statOff:=	di.di_5.bits[4]._inversed,
			
			cmdOn:=		od.do_1.bits[10],
			cmdOff:=	od.do_1.bits[11]
			
		);	
		///////////////////////////////////////////////////////////////////////////////////
		//{name:В3 АВОМ}	
		v3_Avom:Avom3(table:=ADR(imTable)):=(
			statOn:=	di.di_5.bits[5],
			statOff:=	di.di_5.bits[5]._inversed,
			
			cmdOn:=		od.do_1.bits[12],
			cmdOff:=	od.do_1.bits[13]
		);		
		///////////////////////////////////////////////////////////////////////////////////
		//{name:В4 АВОМ}	
		v4_Avom:Avom4(table:=ADR(imTable)):=(
			statOn:=	di.di_5.bits[6],
			statOff:=	di.di_5.bits[6]._inversed,
			
			cmdOn:=		od.do_1.bits[14],
			cmdOff:=	od.do_1.bits[15]
		);	
		///////////////////////////////////////////////////////////////////////////////////
		//{name:ТЭН МБ}	
		TEN_MB:TEN_MB_(table:=ADR(imTable)):=(	
			statOn:=	di.di_10.bits[0],
			statOff:=	di.di_10.bits[0]._inversed,
			
			cmdOn:=		od.do_2.bits[2],
			cmdOff:=	od.do_2.bits[3] 
		);		
		///////////////////////////////////////////////////////////////////////////////////
		//{name:ТЭН Коллектора}	
		TEN_Kollectira:TEN_Kollectora_(table:=ADR(imTable)):=(	
			statOn:=	di.di_10.bits[1],
			statOff:=	di.di_10.bits[1]._inversed,
			
			cmdOn:=		od.do_2.bits[6],
			cmdOff:=	od.do_2.bits[7]
		);		
		///////////////////////////////////////////////////////////////////////////////////
		//{name:ЦМН}	
		CMN:CMN_(table:=ADR(imTable)):=(	
			statOn:=	di.di_10.bits[3],
			statOff:=	di.di_10.bits[3]._inversed,
			
			cmdOn:=		od.do_2.bits[4],
			cmdOff:=	od.do_2.bits[5]
		);		
		///////////////////////////////////////////////////////////////////////////////////
		//{name:ПНС}	
		PNS:PNS_(table:=ADR(imTable)):=(	
			statOn:=	di.di_5.bits[0],
			statOff:=	di.di_5.bits[0]._inversed,
			
			cmdOn:=		od.do_1.bits[0],
			cmdOff:=	od.do_1.bits[1]
		);		
		///////////////////////////////////////////////////////////////////////////////////
		//{name:НУ}
		nu:NasosNu(table:=ADR(imTable)):=(
			nu1:=(	
				statOn:=	di.di_5.bits[1],
				statOff:=	di.di_5.bits[1]._inversed,
				
				cmdOn:=		od.do_1.bits[4],
				cmdOff:=	od.do_1.bits[5]
			),			

			nu2:=(	
				statOn:=	di.di_5.bits[2],
				statOff:=	di.di_5.bits[2]._inversed,
				
				cmdOn:=		od.do_1.bits[6],
				cmdOff:=	od.do_1.bits[7]
			)
				
		);
		///////////////////////////////////////////////////////////////////////////////////
		//{name:Калорифер АВОмасла}
		KaloriferAVOM:Kalorifer_AVOM_(table:=ADR(imTable)):=(	
			statOn:=	di.di_10.bits[2],
			statOff:=	di.di_10.bits[2]._inversed,
			
			cmdOn:=		od.do_2.bits[0],
			cmdOff:=	od.do_2.bits[1]
		);		

		
		
		
		/////////***Дискреты***//////////////////////////////////////////////////////////////////
		///////////Перепад Давления Масло-газ////////////////////////////////////////////////////////////////////////
		//{name:Перепад давления масло-газ  < 100 кПа}
		PerepadDavlenieMasloGaz_Less100:singleSignal(table:=ADR(imTable)):=(signal:=di.di_20.bits[6]);
		//{name:Обрыв сигнала "Перепад давления масло-газ  > 100 кПа"}
		PerepadDavlenieMasloGaz_NS:Reability(table:=ADR(imTable)):=(di1:=di.di_4.bits[0], when:=FALSE);
		//{name:Наличие ЦК "Перепад давления масло-газ  > 100 кПа"}
		PerepadDavlenieMasloGaz_CK:Reability(table:=ADR(imTable)):=(di1:=di.di_4.bits[0], when:=TRUE);	
		
		///////////Перепад На кране 1////////////////////////////////////////////////////////////////////////	
		//{name:Перепад давления на кране 1 < 100 кПа}
		PerepadDavlenieKran1_Less100:singleSignal(table:=ADR(imTable)):=(signal:=di.di_4.bits[1]);
		//{name:Обрыв сигнала "Перепад давления на кране 1 < 100 кПа"}
		PerepadDavlenieKran1_NS:Reability(table:=ADR(imTable)):=(di1:=di.di_4.bits[1], when:=FALSE);
		//{name:Наличие ЦК "Перепад давления на кране 1 < 100 кПа"}
		PerepadDavlenieKran1_CK:Reability(table:=ADR(imTable)):=(di1:=di.di_4.bits[1],  when:=TRUE);
		
		///////////Отклонение уровня масла в аккумуляторе уплотнения////////////////////////////////////////////////////////////////////////
		//{name:Отклонение уровня масла в аккумуляторе уплотнения} 
		LevelMaslaAkkum:ims(table:=ADR(imTable)):=(di1:=di.di_4.bits[2], di2:=di.di_4.bits[2]);
		//{name:Обрыв сигнала "Отклонение уровня масла в аккумуляторе уплотнения"} 
		LevelMaslaAkkum_NS:Reability(table:=ADR(imTable)):=(di1:=di.di_4.bits[2], when:=FALSE);
		//{name:Наличие ЦК "Отклонение уровня масла в аккумуляторе уплотнения"} 
		LevelMaslaAkkum_CK:Reability(table:=ADR(imTable)):=(di1:=di.di_4.bits[2],  when:=TRUE);
		
		///////////Разрешение загрузки двигателя////////////////////////////////////////////////////////////////////////
		//{name:Разрешение загрузки двигателя}
		LoadDriveisGranted:singleSignal(table:=ADR(imTable)):=(signal:=di.di_6.bits[1]);
		//{name:Обрыв сигнала "Разрешение загрузки двигателя"}
		LoadDriveisGranted_NS:Reability(table:=ADR(imTable)):=(di1:=di.di_6.bits[1], when:=FALSE);
		//{name:Наличие ЦК "Разрешение загрузки двигателя"}
		LoadDriveisGranted_CK:Reability(table:=ADR(imTable)):=(di1:=di.di_6.bits[1], when:=TRUE);
		
		///////////Готовность возбудителя////////////////////////////////////////////////////////////////////////
		//{name:Готовность возбудителя}
		VozbutetelisReady:singleSignal(table:=ADR(imTable)):=(signal:=di.di_6.bits[0]);
		//{name:Обрыв сигнала "Готовность возбудителя"}
		VozbutetelisReady_NS :Reability(table:=ADR(imTable)):=(di1:=di.di_6.bits[0], when:=FALSE);
		//{name:Наличие ЦК "Готовность возбудителя"}
		VozbutetelisReady_CK :Reability(table:=ADR(imTable)):=(di1:=di.di_6.bits[0], when:=TRUE);
		
		///////////Неисправность возбудителя////////////////////////////////////////////////////////////////////////
		//{name:Останов по защитам возбудителя (авария)}
		RegVozbOff:singleSignal(table:=ADR(imTable)):=(signal:=di.di_21.bits[7]);
		//{name:Обрыв сигнала "Останов по защитам возбудителя (авария)"}
		RegVozbOff_NS:Reability(table:=ADR(imTable)):=(di1:=di.di_6.bits[2], when:=FALSE);
		//{name:Наличие ЦК  "Останов по защитам возбудителя (авария)"}
		RegVozbOff_CK:Reability(table:=ADR(imTable)):=(di1:=di.di_6.bits[2], when:=TRUE);
		
		///////////Отключение основного регулятора (неисправность)////////////////////////////////////////////////////////////////////////
		//{name:Отключение основного регулятора (неисправность)}
		MainRegOff:singleSignal(table:=ADR(imTable)):=(signal:=di.di_6.bits[3]);
		//{name:Обрыв сигнала "тключение основного регулятора (неисправность)"}
		MainRegOff_NS:Reability(table:=ADR(imTable)):=(di1:=di.di_6.bits[3], when:=FALSE);
		//{name:Наличие ЦК "тключение основного регулятора (неисправность)"}
		MainRegOff_CK:Reability(table:=ADR(imTable)):=(di1:=di.di_6.bits[3], when:=TRUE);
		
		///////////Неисправность цепей управления АВР питания возбудителя////////////////////////////////////////////////////////////////////////
		//{name:Неисправность цепей управления АВР питания возбудителя}
		AVR_Vozb_Malfanctional:singleSignal(table:=ADR(imTable)):=(signal:=di.di_6.bits[4]);
		//{name:Обрыв сигнала "Неисправность цепей управления АВР питания возбудителя"}
		AVR_Vozb_Malfanctional_NS:Reability(table:=ADR(imTable)):=(di1:=di.di_6.bits[4], when:=FALSE);
		//{name:Наличие ЦК "Неисправность цепей управления АВР питания возбудителя"}
		AVR_Vozb_Malfanctional_CK:Reability(table:=ADR(imTable)):=(di1:=di.di_6.bits[4], when:=TRUE);
		
		///////////Аварийное выключение выключателя////////////////////////////////////////////////////////////////////////
		//{name:Аварийное отключение выключателя}
		OFFAvarSwitch:singleSignal(table:=ADR(imTable)):=(signal:=di.di_8.bits[0]);
		//{name:Обрыв сигнала "Аварийное отключение выключателя"}
		OFFAvarSwitch_NS:Reability(table:=ADR(imTable)):=(di1:=di.di_8.bits[0], when:=FALSE);
		//{name:Наличие ЦК "Аварийное отключение выключателя"}
		OFFAvarSwitch_CK:Reability(table:=ADR(imTable)):=(di1:=di.di_8.bits[0], when:=TRUE);
		
		///////////Асинхронный ход перегрузка////////////////////////////////////////////////////////////////////////
		//{name:Асинхронный ход перегрузка}
		AsynchronnyHod:singleSignal(table:=ADR(imTable)):=(signal:=di.di_8.bits[1]);
		//{name:Обрыв сигнала "Асинхронный ход перегрузка"}
		AsynchronnyHod_NS:Reability(table:=ADR(imTable)):=(di1:=di.di_8.bits[1], when:=FALSE);
		//{name:Наличие ЦК  "Асинхронный ход перегрузка"}
		AsynchronnyHod_CK:Reability(table:=ADR(imTable)):=(di1:=di.di_8.bits[1], when:=TRUE);
		
		///////////Автомат в ячейке ШУ включен////////////////////////////////////////////////////////////////////////
		//{name:Автомат в ячейке ШУ включен}
		Avtomat_SHU_on:singleSignal(table:=ADR(imTable)):=(signal:=di.di_8.bits[2]);
		//{name:Обрыв сигнала "Автомат в ячейке ШУ включен"}
		Avtomat_SHU_on_NS:Reability(table:=ADR(imTable)):=(di1:=di.di_8.bits[2], when:=FALSE);
		//{name:Наличие ЦК  "Автомат в ячейке ШУ включен"}
		Avtomat_SHU_on_CK:Reability(table:=ADR(imTable)):=(di1:=di.di_8.bits[2], when:=TRUE);
		
		///////////Автомат в ШП включен////////////////////////////////////////////////////////////////////////
		//{name:Автомат ШП включен}
		Avtomat_SHP_on:singleSignal(table:=ADR(imTable)):=(signal:=di.di_8.bits[3]);
		//{name:Обрыв сигнала "Автомат ШП включен"}
		Avtomat_SHP_on_NS:Reability(table:=ADR(imTable)):=(di1:=di.di_8.bits[3], when:=FALSE);
		//{name:Наличие ЦК "Автомат ШП включен"}
		Avtomat_SHP_on_CK:Reability(table:=ADR(imTable)):=(di1:=di.di_8.bits[3], when:=TRUE);
		
		///////////Напряжение на секции в норме////////////////////////////////////////////////////////////////////////
		//{name:Напряжение на секции в норме}
		U_Sekcii:singleSignal(table:=ADR(imTable)):=(signal:=di.di_8.bits[4]);
		//{name:Обрыв сигнала "Напряжение на секции в норме"}
		U_Sekcii_NS:Reability(table:=ADR(imTable)):=(di1:=di.di_8.bits[4], when:=FALSE);
		//{name:Наличие ЦК "Напряжение на секции в норме"}
		U_Sekcii_CK:Reability(table:=ADR(imTable)):=(di1:=di.di_8.bits[4], when:=TRUE);
		
		///////////Реакторный пуск////////////////////////////////////////////////////////////////////////
		//{name:Реакторный пуск}
		Reactorni_Pusk:singleSignal(table:=ADR(imTable)):=(signal:=di.di_8.bits[5]);
		//{name:Обрыв сигнала "Напряжение на секции в норме"}
		Reactorni_Pusk_NS:Reability(table:=ADR(imTable)):=(di1:=di.di_8.bits[5], when:=FALSE);
		//{name:Наличие ЦК "Напряжение на секции в норме"}
		Reactorni_Pusk_CK:Reability(table:=ADR(imTable)):=(di1:=di.di_8.bits[5], when:=TRUE);
		
		///////////Частотный пуск////////////////////////////////////////////////////////////////////////
		//{name:Частотный пуск}
		Chastotniy_Pusk:singleSignal(table:=ADR(imTable)):=(signal:=di.di_9.bits[0]);
		//{name:Обрыв сигнала "Частотный пуск"}
		Chastotniy_Pusk_NS:Reability(table:=ADR(imTable)):=(di1:=di.di_9.bits[0], when:=FALSE);
		//{name:Наличие ЦК "Частотный пуск"}
		Chastotniy_Pusk_CK:Reability(table:=ADR(imTable)):=(di1:=di.di_9.bits[0], when:=TRUE);
		
		///////////Неуспешный Частотный пуск////////////////////////////////////////////////////////////////////////
		//{name:Неуспешный Частотный пуск}
		Fail_Chastotniy_Pusk:singleSignal(table:=ADR(imTable)):=(signal:=di.di_9.bits[1]);
		//{name:Обрыв сигнала "Неуспешный Частотный пуск"}
		Fail_Chastotniy_Pusk_NS:Reability(table:=ADR(imTable)):=(di1:=di.di_9.bits[1], when:=FALSE);
		//{name:Наличие ЦК "Неуспешный Частотный пуск"}
		Fail_Chastotniy_Pusk_CK:Reability(table:=ADR(imTable)):=(di1:=di.di_9.bits[1], when:=TRUE);
		
		///////////Режим ручного регулирования////////////////////////////////////////////////////////////////////////
		//{name:Режим ручного регулирования}
		Hand_Reg_rej:singleSignal(table:=ADR(imTable)):=(signal:=di.di_9.bits[2]);
		//{name:Обрыв сигнала "Режим ручного регулирования"}
		Hand_Reg_rej_NS:Reability(table:=ADR(imTable)):=(di1:=di.di_9.bits[2], when:=FALSE);
		//{name:Наличие ЦК "Режим ручного регулирования"}
		Hand_Reg_rej_CK:Reability(table:=ADR(imTable)):=(di1:=di.di_9.bits[2], when:=TRUE);
		
